  5254 = 'Warnung active'
  160 = 'Waveform'
  980 = 'Waveform File'
  982 = 'Waveform file'
  983 = 'Waveform req.'
  241 = 'Waveform Update'
  12215 = 'WebStrech calculated'
  1096 = 'WebStrech F. Calc'
  1095 = 'WebStrech F. CANopen'
  1094 = 'WebStrech Factor'
  1093 = 'WebStrech Factor CANopen'
  14157 = 'WebStretchFactor'
  13266 = 'WeuReady'
  6459 = 'wI_NominalSpeed'
  6442 = 'wI_PrintMarkDistance'
  317 = 'wI_PurgeTime'
  318 = 'wI_PurgeWaitTime'
  6465 = 'wI_SheetDetectToMark'
  6425 = 'wI_SheetLength'
  6454 = 'wI_SheetThickness'
  6431 = 'wI_SheetWidth'
  321 = 'wI_WaitValveOn'
  677 = 'Work'
  15392 = 'Worker'
  19928 = 'WorkerCamera'
  4305 = 'WorkerDeformation'
  7307 = 'WorkerDelete'
  4323 = 'WorkerPrint 1'
  9993 = 'WorkerPrint 2'
  8780 = 'WorkerPrint enable'
  10042 = 'WorkerPrint PG: %d'
  6644 = 'WorkerPrint selection: %d'
  2559 = 'WorkerPrint1'
  17071 = 'WorkerPrint2'
  5512 = 'WorkerPrint_fPrintStartOffset'
  13893 = 'WorkerVerify'
  12299 = 'WorkerWeu 1'
  17972 = 'WorkerWeu 2'
  1180 = 'WorkerWeu 3'
  1668 = 'WorkerWeu 4'
  1037 = 'Working distance'
  1040 = 'working distance'
  1041 = 'working range'
  1042 = 'working Tempretaure'
  8216 = 'wO_ConveyorSpeed'
  8231 = 'wO_VarnishQuantity'
  454 = 'WrIdx'
  203 = 'Write'
  1160 = 'Write CSV FILE'
  80 = 'Write Settings'
  350 = 'WriteReq'
  346 = 'WrReq'
  1901 = 'X-Offset'
  154 = 'X-Shift'
  187 = 'X-Shift(Offset)'
  174 = 'X-StartPos'
  886 = 'X0'
  15794 = 'X0: %d'
  1638 = 'x: %0.3f'
  2388 = 'x:%0.3f'
  4503 = 'x=%0.4f'
  6585 = 'x=%d'
  18846 = 'x=%f'
  17127 = 'XD: %d'
  887 = 'XS'
  1122 = 'XShift scaled PG1'
  1123 = 'XShift scaled PG2'
  793 = 'Y Shift'
  3801 = 'Y-Offset'
  1 = 'y-shift'
  155 = 'Y-Shift'
  189 = 'Y-Shift(Offset)'
  5249 = 'y: %0.3f'
  18143 = 'y:%0.3f'
  4527 = 'y=%0.4f'
  16177 = 'y=%d'
  8737 = 'y=%f'
  4637 = 'Zero Balance:'
  542 = 'Zero Scale'
  861 = 'Zoom to caller'
  8214 = '[%%] NeutralFibreFactor'
  6372 = '[%%]NeutralFibreFactor'
  6849 = '[+/-]: %f'
  13426 = '[-] WebStrech calculated'
  4770 = '[-]: %f'
  1136 = '[?]: %f'
  864 = '[Base Speed m/s]: %s'
  111 = '[dpi]: %d'
  865 = '[Factor]: %0.6f'
  103 = '[incr./um]: %0.6f'
  1131 = '[Kp]: %f'
  1097 = '[m/min]: %0.3f'
  1098 = '[m/min]: %f'
  17264 = '[m/s] Max. Speed'
  11491 = '[m/s] Speed'
  409 = '[m/s]: %0.3f'
  10053 = '[m/s]: %0.4f'
  404 = '[m/s]: %0.8f'
  109 = '[m/s]: %f'
  105 = '[mm]: %0.3f'
  434 = '[ms]: %d'
  4812 = '[ms]: %f'
  4403 = '[m]'
  801 = '[m] : %f'
  19619 = '[m] LateralRegister'
  8220 = '[m] Module2ToModule3'
  18328 = '[m] SubstrateLength'
  19359 = '[m] SubstrateThickness'
  118 = '[m]: %f'
  104 = '[pulse/px]: %d'
  119 = '[pulse]: %d'
  9440 = '[Px]'
  416 = '[px]: %d'
  410 = '[p]: %d'
  4778 = '[rev/sec]: %f'
  4795 = '[rev]: %f'
  1128 = '[sec]: %f'
  124 = '[Speed m/s]: %s'
  13566 = '[SubPx]'
  106 = '[SubPx]: %d'
  1133 = '[Tn]: %f'
  856 = '[um/inc]: %0.6f'
  10279 = '[um] : %d'
  1121 = '[um] : %f'
  17520 = '[um] SubstrateThickness'
  6048 = '[] SubstrateThickness'
  12440 = '[µm/inc]: %0.6f'
  6503 = '[µm] SubstrateThickness'
  7367 = '[µm]: %0.6f'
  989 = '[µm]: %d'
  67 = '|'
  16114 = '|- verbose'
  11898 = '|- verbose Mode'
  185 = 'µm: %d'
END_TEXTLIST

// ---- POUs/Products/Ink/InkCirculation/_VISU_InkCirculation.TcVIS
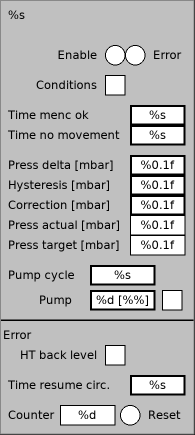
VISUALIZATION _VISU_InkCirculation  // 195x435
VAR_IN_OUT
  m_Inst_Fb : FB_InkCirculation;               (*visu fb instance*) 
END_VAR
    Rectangle (0,0 195x320)
    Rectangle (5,5 180x20), "%s", text variable: m_Inst_Fb._sName
    Ellipse (105,45 20x20), colour toggle: m_Inst_Fb.IbEnable
        toggle m_Inst_Fb.IbEnable
    Rectangle (10,45 90x20), "Enable"
    Ellipse (125,45 20x20), colour toggle: m_Inst_Fb.bLevelError, invisible if: NOT m_Inst_Fb.bLevelError
        toggle m_Inst_Fb.bLevelError
    Rectangle (150,45 40x20), "Error", invisible if: NOT m_Inst_Fb.bLevelError
    Rectangle (5,155 120x20), "Press delta [mbar]"
    Rectangle (130,155 55x20), "%0.1f", text variable: m_Inst_Fb.fRSubMencDeltaP
        OnMouseDown: write the text variable via Edit, min -20, max 0
    Rectangle (5,215 120x20), "Press actual [mbar]"
    Rectangle (130,215 55x20), "%0.1f", text variable: m_Inst_Fb.fSubMencActValue
    Rectangle (5,235 120x20), "Press target [mbar]"
    Rectangle (130,235 55x20), "%0.1f", text variable: m_Inst_Fb.fSubMencTargetValue
    RoundedRectangle (162,290 20x20), colour toggle: m_Inst_Fb.bPumpActivation
    Rectangle (25,290 50x20), "Pump"
    RoundedRectangle (105,75 20x20), colour toggle: m_Inst_Fb.bConditionsMet
    Rectangle (10,75 90x20), "Conditions"
    Rectangle (5,175 120x20), "Hysteresis [mbar]"
    Rectangle (130,175 55x20), "%0.1f", text variable: m_Inst_Fb.fRSubMencHysteresisP
        OnMouseDown: write the text variable via Edit, min 0, max 5
    Rectangle (5,105 120x20), "Time menc ok"
    Rectangle (130,105 55x20), "%s", text variable: m_Inst_Fb.tRSubMencOk
        OnMouseDown: write the text variable via Edit
    Rectangle (5,125 120x20), "Time no movement"
    Rectangle (130,125 55x20), "%s", text variable: m_Inst_Fb.tRNoMovement
        OnMouseDown: write the text variable via Edit
    Rectangle (0,320 195x115)
    Rectangle (0,325 90x20), "Error"
    RoundedRectangle (105,345 20x20), colour toggle: m_Inst_Fb.IbInkLevelReachedBack
    Rectangle (10,345 90x20), "HT back level"
    Rectangle (5,375 120x20), "Time resume circ."
    Rectangle (130,375 55x20), "%s", text variable: m_Inst_Fb.tRResumeCirculation
        OnMouseDown: write the text variable via Edit
    Rectangle (5,405 60x20), "Counter"
    Rectangle (60,405 55x20), "%d", text variable: m_Inst_Fb.nRErrorCounter
    Ellipse (120,405 20x20)
        tap m_Inst_Fb.bResetErrorCounter
    Rectangle (145,405 45x20), "Reset"
    Rectangle (5,195 120x20), "Correction [mbar]"
    Rectangle (130,195 55x20), "%0.1f", text variable: m_Inst_Fb.fRSubMencCorrectionP
        OnMouseDown: write the text variable via Edit, min -1, max 1
    Rectangle (5,265 80x20), "Pump cycle"
    Rectangle (90,265 65x20), "%s", text variable: m_Inst_Fb.tRPumpDutyCycleFrequency
        OnMouseDown: write the text variable via Edit
    Rectangle (90,290 65x20), "%d [%%]", text variable: m_Inst_Fb.nRPumpDutyCycle
        OnMouseDown: write the text variable via Edit
END_VISUALIZATION

// ---- POUs/Products/Machine/_VISU_FUSE_CONTROL.TcVIS
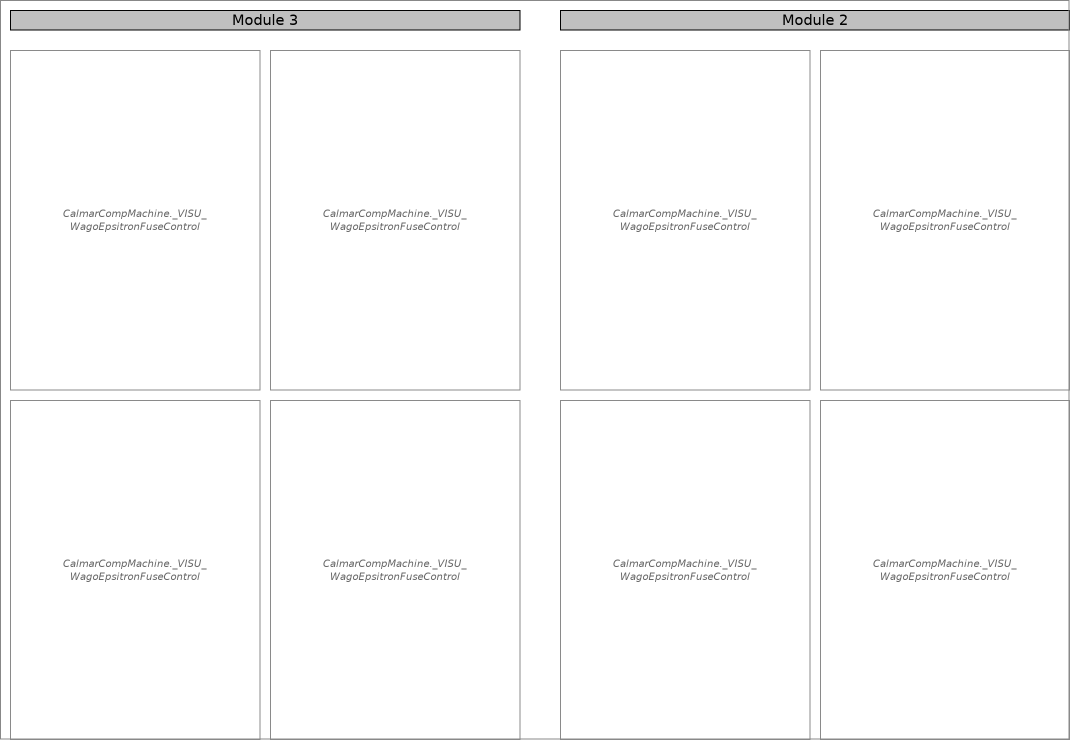
VISUALIZATION _VISU_FUSE_CONTROL  // 1070x740
VAR_IN_OUT
	mInst : FB_WeuPowerControl;
END_VAR
    Frame (820,50 250x340)
        shows CalmarCompMachine._VISU_WagoEpsitronFuseControl(m_Inst_Fb := PRG_MACHINE.fbPowerControl.fb_EpsitronFuseControlF70M1)
    Frame (560,50 250x340)
        shows CalmarCompMachine._VISU_WagoEpsitronFuseControl(m_Inst_Fb := PRG_MACHINE.fbPowerControl.fb_EpsitronFuseControlF90M1)
    Frame (270,50 250x340)
        shows CalmarCompMachine._VISU_WagoEpsitronFuseControl(m_Inst_Fb := PRG_MACHINE.fbPowerControl.fb_EpsitronFuseControlF70M2)
    Frame (10,50 250x340)
        shows CalmarCompMachine._VISU_WagoEpsitronFuseControl(m_Inst_Fb := PRG_MACHINE.fbPowerControl.fb_EpsitronFuseControlF90M2)
    Frame (270,400 250x340), invisible if: TRUE
        shows CalmarCompMachine._VISU_WagoEpsitronFuseControl(m_Inst_Fb := PRG_MACHINE.fbPowerControl.fb_EpsitronFuseControlF122M2)
    Frame (10,400 250x340), invisible if: TRUE
        shows CalmarCompMachine._VISU_WagoEpsitronFuseControl(m_Inst_Fb := PRG_MACHINE.fbPowerControl.fb_EpsitronFuseControlF160M2)
    Frame (820,400 250x340), invisible if: TRUE
        shows CalmarCompMachine._VISU_WagoEpsitronFuseControl(m_Inst_Fb := PRG_MACHINE.fbPowerControl.fb_EpsitronFuseControlF122M1)
    Frame (560,400 250x340), invisible if: TRUE
        shows CalmarCompMachine._VISU_WagoEpsitronFuseControl(m_Inst_Fb := PRG_MACHINE.fbPowerControl.fb_EpsitronFuseControlF160M1)
    Rectangle (10,10 510x20), "Module 3"
    Rectangle (560,10 510x20), "Module 2"
END_VISUALIZATION

// ---- POUs/Products/obsolete/_VISU_DRIFTCONTROL.TcVIS
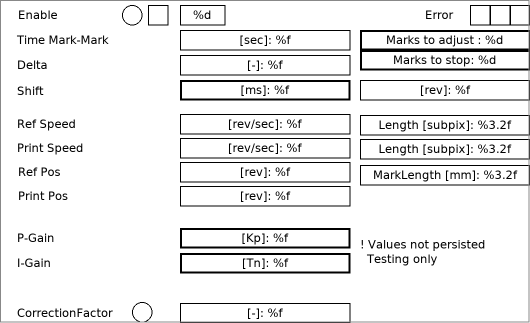
VISUALIZATION _VISU_DRIFTCONTROL  // 530x323
VAR_IN_OUT
  mRef  : FB_DRIFTCONTROL;
END_VAR
    Rectangle (15,5 97x20), "Enable"
    RoundedRectangle (148,5 20x20), colour toggle: mRef.bL_ControlActive
    Ellipse (122,5 20x20), colour toggle: mRef.bI_Enable
        toggle mRef.bI_Enable
    Rectangle (14,30 120x20), "Time Mark-Mark"
    Rectangle (180,30 170x20), "[sec]: %f", text variable: mRef.fL_DeltaTimeStamp
    Rectangle (14,55 120x20), "Delta"
    Rectangle (180,55 170x20), "[-]: %f", text variable: mRef.fL_DeltaCtrl
    Rectangle (14,228 120x20), "P-Gain"
    Rectangle (180,228 170x20), "[Kp]: %f", text variable: mRef.fI_ControllerPGain
        OnMouseDown: write the text variable via Default
    Rectangle (14,253 120x20), "I-Gain"
    Rectangle (180,253 170x20), "[Tn]: %f", text variable: mRef.fI_ControllerIGain
        OnMouseDown: write the text variable via Edit
    Rectangle (14,303 120x20), "CorrectionFactor"
    Rectangle (180,303 170x20), "[-]: %f", text variable: mRef.fO_SpeedCorrectionFactor
    Rectangle (14,114 120x20), "Ref Speed"
    Rectangle (180,114 170x20), "[rev/sec]: %f", text variable: mRef.fL_RefSpeed
    Rectangle (14,138 120x20), "Print Speed"
    Rectangle (180,138 170x20), "[rev/sec]: %f", text variable: mRef.fL_ImgSpeed
    Ellipse (132,302 20x20), colour toggle: mRef.bI_OutputEnable
        toggle mRef.bI_OutputEnable
    Rectangle (360,115 170x20), "Length [subpix]: %3.2f", text variable: mRef.fL_RefLength, colour toggle: mRef.bL_FormatWarning
    Rectangle (360,139 170x20), "Length [subpix]: %3.2f", text variable: mRef.lL_ImgLength, colour toggle: mRef.bL_FormatWarning
    Rectangle (15,162 120x20), "Ref Pos"
    Rectangle (180,162 170x20), "[rev]: %f", text variable: mRef.fL_RefPos
    Rectangle (15,186 120x20), "Print Pos"
    Rectangle (180,186 170x20), "[rev]: %f", text variable: mRef.fL_ImgPos
    RoundedRectangle (470,5 20x20), tooltip "ctrl err", colour toggle: mRef.bO_ContrErr
        tap mRef.bL_ResetInternal
    Rectangle (422,5 42x20), "Error"
    Rectangle (357,233 141x38), "! Values not persisted Testing only"
    Rectangle (180,80 170x20), "[ms]: %f", text variable: mRef.fI_DriftTimeShift
        OnMouseDown: write the text variable via Default
    Rectangle (14,81 120x20), "Shift"
    Rectangle (360,80 170x20), "[rev]: %f", text variable: mRef.fL_ShiftPos
    Rectangle (180,5 45x20), "%d", text variable: mRef.iL_State
    RoundedRectangle (490,5 20x20), tooltip "fb err", colour toggle: mRef.bL_Error
        tap mRef.bL_ResetInternal
    RoundedRectangle (510,5 20x20), tooltip "arw", colour toggle: mRef.fL_CtrlGainFactor <> 1
        tap mRef.bL_ResetInternal
    Rectangle (360,165 170x20), "MarkLength [mm]: %3.2f", text variable: mRef.fL_RefLengthMM, colour toggle: mRef.bL_FormatWarning
    Rectangle (360,30 170x20), "Marks to adjust : %d", text variable: mRef.nI_NbCyclesToAdjust, colour toggle: mRef.bO_ControllerAdjusted
        OnMouseDown: write the text variable via Default
    Rectangle (360,50 170x20), "Marks to stop: %d", text variable: mRef.nI_NbMissMarksToStop, colour toggle: mRef.bO_ControllerAdjusted
        OnMouseDown: write the text variable via Default
END_VISUALIZATION

// ---- POUs/Products/Print_Weu/Mark/_VISU_CameraTrigger.TcVIS
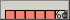
VISUALIZATION _VISU_CameraTrigger  // 70x20
VAR_IN_OUT
	mInst : FB_MarkDetection;
END_VAR
    RoundedRectangle (0,0 70x20), tooltip "Trigger Armed", colour toggle: mInst.bTriggerArmed
    RoundedRectangle (15,10 10x10), tooltip "Speed valid", colour toggle: mInst.bSpeedValid
    RoundedRectangle (25,10 10x10), tooltip "Cam valid", colour toggle: mInst.bCamValid
    RoundedRectangle (35,10 10x10), tooltip "marks valid", colour toggle: mInst.bMarkValid
    RoundedRectangle (5,10 10x10), tooltip "Init ok", colour toggle: mInst.bInitOk
    Rectangle (0,0 70x10), tooltip "Trigger active"
    RoundedRectangle (55,10 10x10), "%d", tooltip "e state", text variable: mInst.nMarkSelection
    RoundedRectangle (45,10 10x10), tooltip "(Hw)Enable", colour toggle: mInst.bEnable
END_VISUALIZATION

// ---- POUs/Products/Print_Weu/Mark/_VISU_MarkCamera_WEU.TcVIS
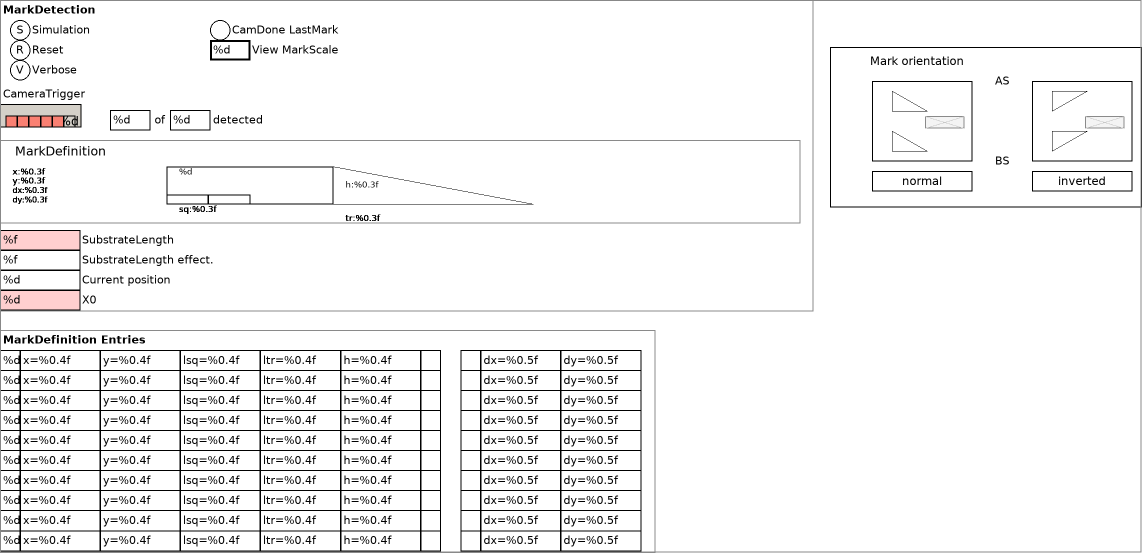
VISUALIZATION _VISU_MarkCamera_WEU  // 1142x553
VAR_IN_OUT
  mCam : FB_MarkCamera_WEU;
  mMarkDetect : FB_MarkDetection;
END_VAR
    Frame (0,330 655x223)
        shows _VISU_MarkDefinition(mInst := mMarkDetect._pFbMarkDefinition^)
    Frame (0,0 813x311)
        shows _VISU_MarkDetection(mInst := mMarkDetect)
    Rectangle (830,47 312x160)
    Rectangle (867,51 124x20), "Mark orientation"
    Rectangle (872,81 100x80)
    Polygon (892,91) (892,111) (927,111)
    Polygon (892,131) (892,151) (927,151)
    Image (925,116 39x12), image: VisuSymbols.Symbols.ArrowBoldLeft
    Rectangle (992,71 25x20), "AS"
    Rectangle (992,151 25x20), "BS"
    Rectangle (1032,81 100x80)
    Polygon (1052,91) (1052,111) (1087,91)
    Polygon (1052,131) (1052,151) (1087,131)
    Image (1085,116 39x12), image: VisuSymbols.Symbols.ArrowBoldLeft
    RoundedRectangle (872,171 100x20), "normal"
    RoundedRectangle (1032,171 100x20), "inverted"
END_VISUALIZATION

// ---- POUs/Products/Print_Weu/Mark/_VISU_MarkDefinition.TcVIS
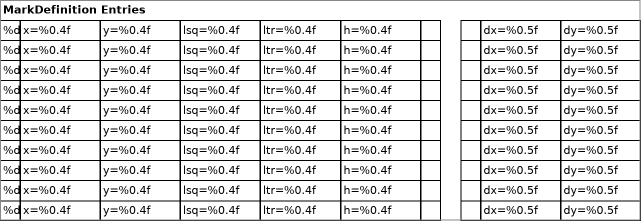
VISUALIZATION _VISU_MarkDefinition  // 641x221
VAR_IN_OUT
	mInst : FB_MarkDefinition;
END_VAR
    Rectangle (0,0 159x20), "MarkDefinition Entries"
    Frame (0,20 641x21)
        shows _VISU_MarkTriangle_Detail(mInst := mInst.sMarkDef[1])
    Frame (0,40 641x21)
        shows _VISU_MarkTriangle_Detail(mInst := mInst.sMarkDef[2])
    Frame (0,60 641x21)
        shows _VISU_MarkTriangle_Detail(mInst := mInst.sMarkDef[3])
    Frame (0,80 641x21)
        shows _VISU_MarkTriangle_Detail(mInst := mInst.sMarkDef[4])
    Frame (0,100 641x21)
        shows _VISU_MarkTriangle_Detail(mInst := mInst.sMarkDef[5])
    Frame (0,200 641x21)
        shows _VISU_MarkTriangle_Detail(mInst := mInst.sMarkDef[10])
    Frame (0,120 641x21)
        shows _VISU_MarkTriangle_Detail(mInst := mInst.sMarkDef[6])
    Frame (0,140 641x21)
        shows _VISU_MarkTriangle_Detail(mInst := mInst.sMarkDef[7])
    Frame (0,160 641x21)
        shows _VISU_MarkTriangle_Detail(mInst := mInst.sMarkDef[8])
    Frame (0,180 641x21)
        shows _VISU_MarkTriangle_Detail(mInst := mInst.sMarkDef[9])
END_VISUALIZATION

// ---- POUs/Products/Print_Weu/Mark/_VISU_MarkDefinition_View.TcVIS
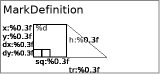
VISUALIZATION _VISU_MarkDefinition_View  // 160x74
VAR_IN_OUT
	mInst : FB_MarkDefinition;
  xScale : UDINT;
END_VAR
    Frame (0,24 160x50), invisible if: NOT mInst.sMarkDef[1].bShow
        shows _VISU_MarkTriangle(mInst := mInst.sMarkDef[1])
        p3560616238: mInst.sMarkDef[1].nMove*xScale
    Frame (0,24 160x50), invisible if: NOT mInst.sMarkDef[2].bShow
        shows _VISU_MarkTriangle(mInst := mInst.sMarkDef[2])
        p3560616238: mInst.sMarkDef[2].nMove*xScale
    Frame (0,24 160x50), invisible if: NOT mInst.sMarkDef[3].bShow
        shows _VISU_MarkTriangle(mInst := mInst.sMarkDef[3])
        p3560616238: mInst.sMarkDef[3].nMove*xScale
    Frame (0,24 160x50), invisible if: NOT mInst.sMarkDef[6].bShow
        shows _VISU_MarkTriangle(mInst := mInst.sMarkDef[6])
        p3560616238: mInst.sMarkDef[6].nMove*xScale
    Frame (0,24 160x50), invisible if: NOT mInst.sMarkDef[4].bShow
        shows _VISU_MarkTriangle(mInst := mInst.sMarkDef[4])
        p3560616238: mInst.sMarkDef[4].nMove*xScale
    Frame (0,24 160x50), invisible if: NOT mInst.sMarkDef[5].bShow
        shows _VISU_MarkTriangle(mInst := mInst.sMarkDef[5])
        p3560616238: mInst.sMarkDef[5].nMove*xScale
    Frame (0,24 160x50), invisible if: NOT mInst.sMarkDef[7].bShow
        shows _VISU_MarkTriangle(mInst := mInst.sMarkDef[7])
        p3560616238: mInst.sMarkDef[7].nMove*xScale
    Frame (0,24 160x50), invisible if: NOT mInst.sMarkDef[10].bShow
        shows _VISU_MarkTriangle(mInst := mInst.sMarkDef[10])
        p3560616238: mInst.sMarkDef[10].nMove*xScale
    Frame (0,24 160x50), invisible if: NOT mInst.sMarkDef[8].bShow
        shows _VISU_MarkTriangle(mInst := mInst.sMarkDef[8])
        p3560616238: mInst.sMarkDef[8].nMove*xScale
    Frame (0,24 160x50), invisible if: NOT mInst.sMarkDef[9].bShow
        shows _VISU_MarkTriangle(mInst := mInst.sMarkDef[9])
        p3560616238: mInst.sMarkDef[9].nMove*xScale
    Rectangle (0,0 120x20), "MarkDefinition"
END_VISUALIZATION

// ---- POUs/Products/Print_Weu/Mark/_VISU_MarkDefinition_View_edit.TcVIS
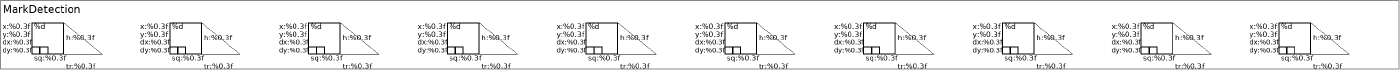
VISUALIZATION _VISU_MarkDefinition_View_edit  // 1463x74
VAR_IN_OUT
	mInst : FB_MarkDefinition;
  xScale : UDINT;
END_VAR
    Frame (0,24 160x50), invisible if: NOT mInst.sMarkDef[1].bShow
        shows _VISU_MarkTriangle(mInst := mInst.sMarkDef[1])
    Frame (144,24 160x50), invisible if: NOT mInst.sMarkDef[2].bShow
        shows _VISU_MarkTriangle(mInst := mInst.sMarkDef[2])
    Frame (289,24 160x50), invisible if: NOT mInst.sMarkDef[3].bShow
        shows _VISU_MarkTriangle(mInst := mInst.sMarkDef[3])
    Frame (724,24 160x50), invisible if: NOT mInst.sMarkDef[6].bShow
        shows _VISU_MarkTriangle(mInst := mInst.sMarkDef[6])
    Frame (434,24 160x50), invisible if: NOT mInst.sMarkDef[4].bShow
        shows _VISU_MarkTriangle(mInst := mInst.sMarkDef[4])
    Frame (579,24 160x50), invisible if: NOT mInst.sMarkDef[5].bShow
        shows _VISU_MarkTriangle(mInst := mInst.sMarkDef[5])
    Frame (869,24 160x50), invisible if: NOT mInst.sMarkDef[7].bShow
        shows _VISU_MarkTriangle(mInst := mInst.sMarkDef[7])
    Frame (1303,24 160x50), invisible if: NOT mInst.sMarkDef[10].bShow
        shows _VISU_MarkTriangle(mInst := mInst.sMarkDef[10])
    Frame (1014,24 160x50), invisible if: NOT mInst.sMarkDef[8].bShow
        shows _VISU_MarkTriangle(mInst := mInst.sMarkDef[8])
    Frame (1159,24 160x50), invisible if: NOT mInst.sMarkDef[9].bShow
        shows _VISU_MarkTriangle(mInst := mInst.sMarkDef[9])
    Rectangle (0,0 120x20), "MarkDetection"
END_VISUALIZATION

// ---- POUs/Products/Print_Weu/Mark/_VISU_MarkDetection.TcVIS
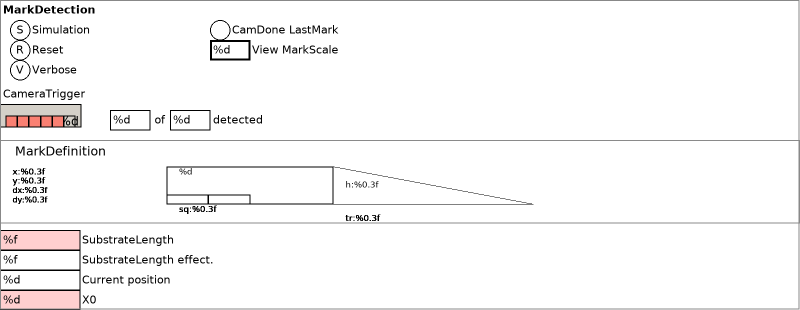
VISUALIZATION _VISU_MarkDetection  // 800x310
VAR_IN_OUT
	mInst: FB_MarkDetection;
END_VAR
    Rectangle (0,0 120x20), "MarkDetection"
    Rectangle (170,110 40x20), "%d", tooltip "teached marks", text variable: mInst._pFbMarkDefinition^._nMarks, colour toggle: mInst._pFbMarkDefinition^._nMarks = 0
    Rectangle (110,110 40x20), "%d", tooltip "detected marks", text variable: mInst._pFbMarkDefinition^._nMarksDetected, colour toggle: mInst._pFbMarkDefinition^._nMarksDetected >= mInst._pFbMarkDefinition^._nMarks AND mInst._pFbMarkDefinition^._nMarks > 0
    Ellipse (10,40 20x20), "R", tooltip "Reset"
        tap mInst.bManualReset
    Frame (0,104 81x26)
        shows _VISU_CameraTrigger(mInst := mInst)
    Rectangle (0,84 120x20), "CameraTrigger"
    Rectangle (210,110 60x20), "detected"
    Rectangle (150,110 20x20), "of"
    Rectangle (0,230 80x20), "%f", text variable: mInst._fSubstrateLength, colour toggle: mInst._fSubstrateLength > 0
    Rectangle (79,230 140x20), "SubstrateLength"
    Rectangle (0,250 80x20), "%f", text variable: mInst._fSubstrateLengthEffective
    Rectangle (79,250 140x20), "SubstrateLength effect."
    Rectangle (0,290 80x20), "%d", text variable: mInst._nX0, colour toggle: mInst._bValid
    Rectangle (79,290 140x20), "X0"
    Rectangle (0,270 80x20), "%d", text variable: mInst.nCurrentPos
    Rectangle (79,270 140x20), "Current position"
    Frame (0,140 800x83)
        shows _VISU_MarkDefinition_View(mInst := mInst._pFbMarkDefinition^, xScale := mInst.nMarkXMoveScale)
    Ellipse (10,20 20x20), "S", tooltip "Simulation"
        toggle mInst._bSimEnable
    Rectangle (29,20 140x20), "Simulation"
    Ellipse (210,20 20x20)
        toggle mInst.bR_TerminateLast
    Rectangle (229,20 140x20), "CamDone LastMark"
    Rectangle (210,40 40x20), "%d", text variable: mInst.nMarkXMoveScale
        OnMouseClick: write the text variable via Default
    Rectangle (249,40 100x20), "View MarkScale"
    Rectangle (29,40 140x20), "Reset"
    Ellipse (10,60 20x20), "V", tooltip "Verbose"
        toggle mInst._bVerbose
    Rectangle (29,60 140x20), "Verbose"
END_VISUALIZATION

// ---- POUs/Products/Print_Weu/Mark/_VISU_MarkTriangle.TcVIS
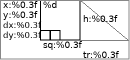
VISUALIZATION _VISU_MarkTriangle  // 130x60
VAR_IN_OUT
	mInst : ST_MarkDefinition;
END_VAR
    Rectangle (40,0 40x40), colour toggle: mInst.sState.bSet
        p874137650: mInst.fSqLength/mInst.fHeight*40-40
    Polygon (80,0) (80,40) (128,40), colour toggle: mInst.sState.bSet
        p3560616238: mInst.fSqLength/mInst.fHeight*40-40
    Rectangle (80,9 40x20), "h:%0.3f", tooltip "[m]", text variable: mInst.fHeight
        p3560616238: mInst.fSqLength/mInst.fHeight*40-40
    Rectangle (80,50 50x10), "tr:%0.3f", tooltip "[m]", text variable: mInst.fTrLength
        p3560616238: mInst.fSqLength/mInst.fHeight*40-40
    Rectangle (40,40 50x10), "sq:%0.3f", tooltip "[m]", text variable: mInst.fSqLength
    Rectangle (40,0 30x10), "%d", tooltip "Id", text variable: mInst.nId
    Rectangle (0,0 40x10), "x:%0.3f", tooltip "[m]", text variable: mInst.fPosX
    Rectangle (0,10 40x10), "y:%0.3f", tooltip "[m]", text variable: mInst.fPosY
    RoundedRectangle (40,30 10x10), tooltip "Missed", colour toggle: mInst.sState.bMissed, invisible if: NOT mInst.sState.bSet
    RoundedRectangle (50,30 10x10), tooltip "InArea", colour toggle: mInst.sState.bInArea, invisible if: NOT mInst.sState.bSet
    Rectangle (0,20 40x10), "dx:%0.3f", tooltip "[m]", text variable: mInst.sState.dx, invisible if: NOT mInst.sState.bSet
    Rectangle (0,30 40x10), "dy:%0.3f", tooltip "[m]", text variable: mInst.sState.dy, invisible if: NOT mInst.sState.bSet
END_VISUALIZATION

// ---- POUs/Products/Print_Weu/Mark/_VISU_MarkTriangle_Detail.TcVIS
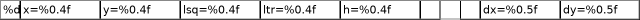
VISUALIZATION _VISU_MarkTriangle_Detail  // 640x20
VAR_IN_OUT
	mInst : ST_MarkDefinition;
END_VAR
    Rectangle (20,0 80x20), "x=%0.4f", text variable: mInst.fPosX
        OnMouseClick: write the text variable via Default
    Rectangle (100,0 80x20), "y=%0.4f", text variable: mInst.fPosY
        OnMouseClick: write the text variable via Default
    RoundedRectangle (460,0 20x20)
        toggle mInst.sState.bSet
    Rectangle (480,0 80x20), "dx=%0.5f", text variable: minst.sState.dx
        OnMouseClick: write the text variable via Default
    Rectangle (560,0 80x20), "dy=%0.5f", text variable: minst.sState.dy
        OnMouseClick: write the text variable via Default
    Rectangle (0,0 20x20), "%d", text variable: mInst.nId, colour toggle: mInst.nId > 0
    RoundedRectangle (420,0 20x20), tooltip "inverted X"
        toggle mInst.bInvertedX
    Rectangle (260,0 80x20), "ltr=%0.4f", text variable: mInst.fTrLength
        OnMouseClick: write the text variable via Default
    Rectangle (340,0 80x20), "h=%0.4f", text variable: mInst.fHeight
        OnMouseClick: write the text variable via Default
    Rectangle (180,0 80x20), "lsq=%0.4f", text variable: mInst.fSqLength
        OnMouseClick: write the text variable via Default
END_VISUALIZATION

// ---- POUs/Products/Print_Weu/UV_LED_Modul/_VISU_UvLedModule.TcVIS
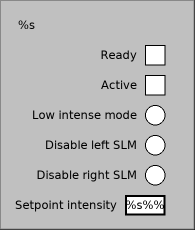
VISUALIZATION _VISU_UvLedModule  // 195x230
VAR_IN_OUT
  m_Inst_Fb   : FB_UvLedModule;
END_VAR
    Rectangle (0,0 195x230), colour variable: m_Inst_Fb._StInkDefinition.lI_ColorRGB
        p2167032090: m_Inst_Fb._StInkDefinition.lI_ColorRGB
        p3092690914: 16#FFFF0000
        p3450524324: 16#FF000000
    Rectangle (15,15 155x20), "%s", text variable: m_Inst_Fb._StInkDefinition.aI_ColorName
    RoundedRectangle (145,45 20x20), colour toggle: m_Inst_Fb.IbReady
    Rectangle (20,45 120x20), "Ready"
    RoundedRectangle (145,75 20x20), colour toggle: m_Inst_Fb._bActivate
    Rectangle (20,75 120x20), "Active"
    Ellipse (145,105 20x20), colour toggle: m_Inst_Fb.RbLowIntenseMode
        toggle m_Inst_Fb.RbLowIntenseMode
    Rectangle (20,105 120x20), "Low intense mode"
    Ellipse (145,135 20x20), colour toggle: m_Inst_Fb.RbDisableLeft
        toggle m_Inst_Fb.RbDisableLeft
    Rectangle (20,135 120x20), "Disable left SLM"
    Ellipse (145,165 20x20), colour toggle: m_Inst_Fb.RbDisableRight
        toggle m_Inst_Fb.RbDisableRight
    Rectangle (20,165 120x20), "Disable right SLM"
    Rectangle (11,195 109x20), "Setpoint intensity"
    Rectangle (125,195 40x20), "%s%%", text variable: m_Inst_Fb.RnIntensitySetpoint
        OnMouseDown: write the text variable via VisuDialogs.Numpad, min m_Inst_Fb.CnMinIntensitySetpoint, max m_Inst_Fb.CnMaxIntensitySetpoint
END_VISUALIZATION

// ---- POUs/Products/Print_Weu/VISU_PAPER_POS_DETECT.TcVIS
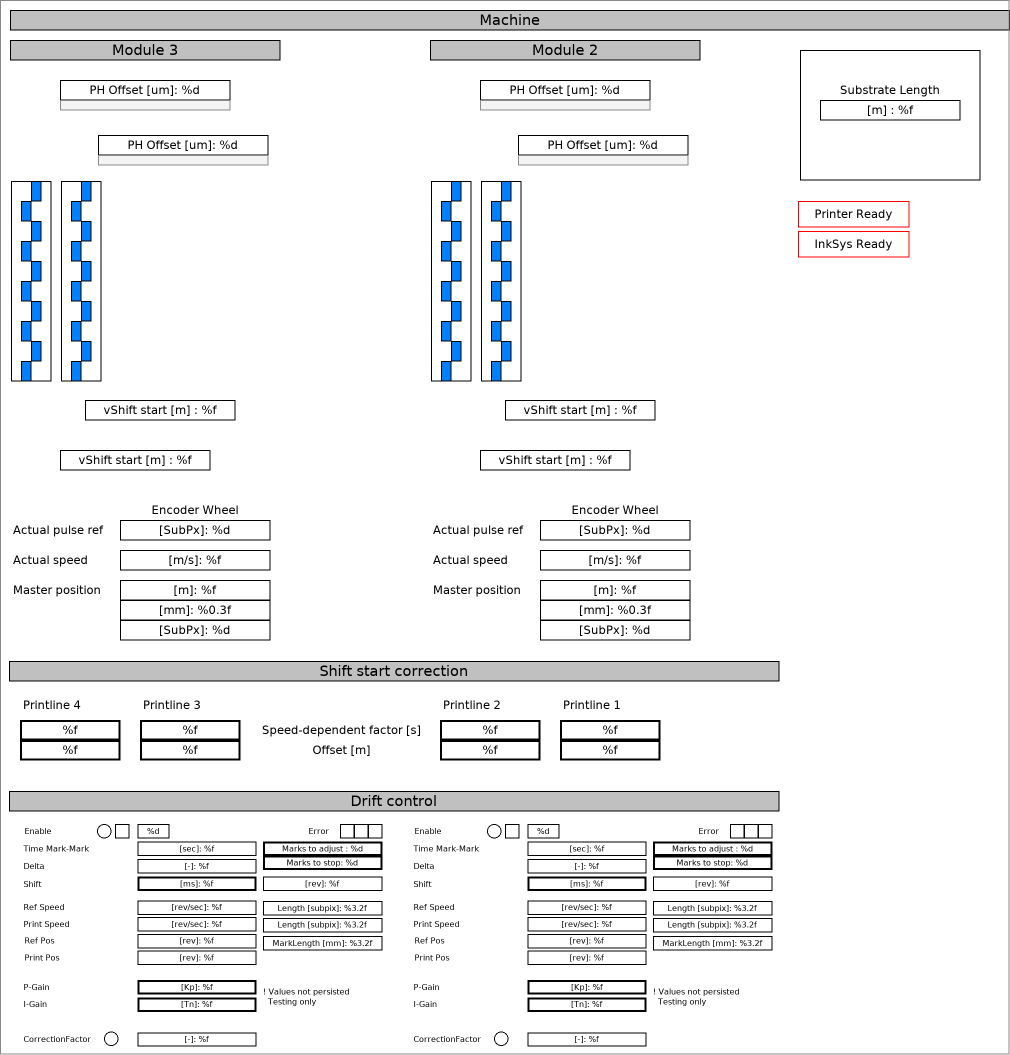
VISUALIZATION VISU_PAPER_POS_DETECT  // 1010x1055
    Polyline (100,340)
    Rectangle (800,50 180x130)
    Rectangle (10,10 1000x20), "Machine"
    Rectangle (820,100 140x20), "[m] : %f", text variable: PRG_PRINT.fL_SubstrateLen[ePr_PG_GROUP_1]
        OnMouseDown: write the text variable via Edit
    Rectangle (820,80 140x20), "Substrate Length"
    Rectangle (798,201 111x26), "Printer Ready", colour toggle: PRG_MACHINE.bO_PrinterReady
    Rectangle (798,231 111x26), "InkSys Ready", colour toggle: PRG_INK.bO_InkSystemOk
    Group (61,181 38x198)
        Rectangle (0,0 40x200)
        Rectangle (20,0 10x20)
        Rectangle (10,20 10x20)
        Rectangle (20,40 10x20)
        Rectangle (10,60 10x20)
        Rectangle (20,80 10x20)
        Rectangle (10,100 10x20)
        Rectangle (20,120 10x20)
        Rectangle (10,140 10x20)
        Rectangle (20,160 10x20)
        Rectangle (10,180 10x20)
    Group (11,181 38x198)
        Rectangle (0,0 40x200)
        Rectangle (20,0 10x20)
        Rectangle (10,20 10x20)
        Rectangle (20,40 10x20)
        Rectangle (10,60 10x20)
        Rectangle (20,80 10x20)
        Rectangle (10,100 10x20)
        Rectangle (20,120 10x20)
        Rectangle (10,140 10x20)
        Rectangle (20,160 10x20)
        Rectangle (10,180 10x20)
    Rectangle (60,80 170x20), "PH Offset [um]: %d", text variable: PRG_PRINT.sAdsPrintGroup[ePr_PG_GROUP_4].sI_ShiftPositionX.lI_Val
        OnMouseDown: write the text variable via Edit
    Scrollbar (60,100 170x10)
        p1057716461: PRG_PRINT.sAdsPrintGroup[ePr_PG_GROUP_2].sI_ShiftPositionX.lI_Val
    Polyline (100,140)
    Polyline (150,360)
    Rectangle (98,135 170x20), "PH Offset [um]: %d", text variable: PRG_PRINT.sAdsPrintGroup[ePr_PG_GROUP_3].sI_ShiftPositionX.lI_Val
        OnMouseDown: write the text variable via Edit
    Scrollbar (98,155 170x10)
        p1057716461: PRG_PRINT.sAdsPrintGroup[ePr_PG_GROUP_1].sI_ShiftPositionX.lI_Val
    Polyline (150,360)
    Polyline (250,350)
    Rectangle (85,400 150x20), "vShift start [m] : %f", text variable: PRG_PRINT.fbWorkerWeu[3].fPosition
    Rectangle (60,450 150x20), "vShift start [m] : %f", text variable: PRG_PRINT.fbWorkerWeu[4].fPosition
    Polyline (100,340)
    Group (481,181 38x198)
        Rectangle (0,0 40x200)
        Rectangle (20,0 10x20)
        Rectangle (10,20 10x20)
        Rectangle (20,40 10x20)
        Rectangle (10,60 10x20)
        Rectangle (20,80 10x20)
        Rectangle (10,100 10x20)
        Rectangle (20,120 10x20)
        Rectangle (10,140 10x20)
        Rectangle (20,160 10x20)
        Rectangle (10,180 10x20)
    Group (431,181 38x198)
        Rectangle (0,0 40x200)
        Rectangle (20,0 10x20)
        Rectangle (10,20 10x20)
        Rectangle (20,40 10x20)
        Rectangle (10,60 10x20)
        Rectangle (20,80 10x20)
        Rectangle (10,100 10x20)
        Rectangle (20,120 10x20)
        Rectangle (10,140 10x20)
        Rectangle (20,160 10x20)
        Rectangle (10,180 10x20)
    Rectangle (480,80 170x20), "PH Offset [um]: %d", text variable: PRG_PRINT.sAdsPrintGroup[ePr_PG_GROUP_2].sI_ShiftPositionX.lI_Val
        OnMouseDown: write the text variable via Edit
    Scrollbar (480,100 170x10)
        p1057716461: PRG_PRINT.sAdsPrintGroup[ePr_PG_GROUP_2].sI_ShiftPositionX.lI_Val
    Polyline (100,140)
    Polyline (150,360)
    Rectangle (518,135 170x20), "PH Offset [um]: %d", text variable: PRG_PRINT.sAdsPrintGroup[ePr_PG_GROUP_1].sI_ShiftPositionX.lI_Val
        OnMouseDown: write the text variable via Edit
    Scrollbar (518,155 170x10)
        p1057716461: PRG_PRINT.sAdsPrintGroup[ePr_PG_GROUP_1].sI_ShiftPositionX.lI_Val
    Polyline (150,360)
    Polyline (250,350)
    Rectangle (505,400 150x20), "vShift start [m] : %f", text variable: PRG_PRINT.fbWorkerWeu[1].fPosition
    Rectangle (480,450 150x20), "vShift start [m] : %f", text variable: PRG_PRINT.fbWorkerWeu[2].fPosition
    Rectangle (10,40 270x20), "Module 3"
    Rectangle (430,40 270x20), "Module 2"
    Rectangle (120,600 150x20), "[mm]: %0.3f", text variable: 0.001*PRG_PRINT.Fb_Ph_Master[ePr_PG_GROUP_2].fO_Master_Position
    Rectangle (120,620 150x20), "[SubPx]: %d", text variable: PRG_PRINT.Fb_Ph_Master[ePr_PG_GROUP_2].lO_Master_Position
    Rectangle (120,550 150x20), "[m/s]: %f", text variable: PRG_PRINT.Fb_Ph_Master[ePr_PG_GROUP_2].fO_Master_Speed
    Rectangle (10,550 100x20), "Actual speed"
    Rectangle (10,580 100x20), "Master position"
    Rectangle (120,520 150x20), "[SubPx]: %d", text variable: PRG_PRINT.Fb_Ph_Master[ePr_PG_GROUP_2].lI_Reference
    Rectangle (10,520 100x20), "Actual pulse ref"
    Rectangle (120,500 150x20), "Encoder Wheel"
    Rectangle (120,580 150x20), "[m]: %f", text variable: 0.000001*PRG_PRINT.Fb_Ph_Master[ePr_PG_GROUP_2].fO_Master_Position
    Rectangle (540,600 150x20), "[mm]: %0.3f", text variable: 0.001*PRG_PRINT.Fb_Ph_Master[ePr_PG_GROUP_1].fO_Master_Position
    Rectangle (540,620 150x20), "[SubPx]: %d", text variable: PRG_PRINT.Fb_Ph_Master[ePr_PG_GROUP_1].lO_Master_Position
    Rectangle (540,550 150x20), "[m/s]: %f", text variable: PRG_PRINT.Fb_Ph_Master[ePr_PG_GROUP_1].fO_Master_Speed
    Rectangle (430,550 100x20), "Actual speed"
    Rectangle (430,580 100x20), "Master position"
    Rectangle (540,520 150x20), "[SubPx]: %d", text variable: PRG_PRINT.Fb_Ph_Master[ePr_PG_GROUP_1].lI_Reference
    Rectangle (430,520 100x20), "Actual pulse ref"
    Rectangle (540,500 150x20), "Encoder Wheel"
    Rectangle (540,580 150x20), "[m]: %f", text variable: 0.000001*PRG_PRINT.Fb_Ph_Master[ePr_PG_GROUP_1].fO_Master_Position
    Frame (12,821 370x234)
        shows _VISU_DRIFTCONTROL(mRef := PRG_PRINT.fB_DriftControl[2])
    Rectangle (9,791 770x20), "Drift control"
    Frame (402,821 370x234)
        shows _VISU_DRIFTCONTROL(mRef := PRG_PRINT.fB_DriftControl[1])
    Rectangle (9,661 770x20), "Shift start correction"
    Rectangle (560,695 100x20), "Printline 1"
    Rectangle (560,720 100x20), "%f", text variable: PRG_PRINT.fbWorkerWeu[1]._fStartShiftFactor
        OnMouseDown: write the text variable via Edit
    Rectangle (560,740 100x20), "%f", text variable: PRG_PRINT.fbWorkerWeu[1]._fStartShiftOffset
        OnMouseDown: write the text variable via Edit
    Rectangle (250,720 180x20), "Speed-dependent factor [s]"
    Rectangle (250,740 180x20), "Offset [m]"
    Rectangle (440,695 100x20), "Printline 2"
    Rectangle (440,720 100x20), "%f", text variable: PRG_PRINT.fbWorkerWeu[2]._fStartShiftFactor
        OnMouseDown: write the text variable via Edit
    Rectangle (440,740 100x20), "%f", text variable: PRG_PRINT.fbWorkerWeu[2]._fStartShiftOffset
        OnMouseDown: write the text variable via Edit
    Rectangle (140,695 100x20), "Printline 3"
    Rectangle (140,720 100x20), "%f", text variable: PRG_PRINT.fbWorkerWeu[3]._fStartShiftFactor
        OnMouseDown: write the text variable via Edit
    Rectangle (140,740 100x20), "%f", text variable: PRG_PRINT.fbWorkerWeu[3]._fStartShiftOffset
        OnMouseDown: write the text variable via Edit
    Rectangle (20,695 100x20), "Printline 4"
    Rectangle (20,720 100x20), "%f", text variable: PRG_PRINT.fbWorkerWeu[4]._fStartShiftFactor
        OnMouseDown: write the text variable via Edit
    Rectangle (20,740 100x20), "%f", text variable: PRG_PRINT.fbWorkerWeu[4]._fStartShiftOffset
        OnMouseDown: write the text variable via Edit
END_VISUALIZATION

// ---- POUs/Products/Print_Weu/_VISU_Templates/_VISU_CT_Details.TcVIS
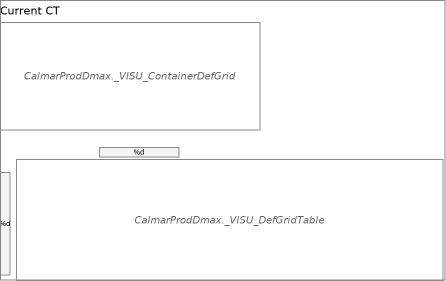
VISUALIZATION _VISU_CT_Details  // 446x281
VAR_IN_OUT
  mInst : FB_WorkerDefGrid_Deformation;
END_VAR
    Frame (0,22 260x108)
        shows CalmarProdDmax._VISU_ContainerDefGrid(m_Inst := mInst._pMultiAttachedCTs[1]^)
    Frame (16,159 427x122)
        shows CalmarProdDmax._VISU_DefGridTable(m_Inst := mInst._pMultiAttachedCTs[1]^.fBImageDeformation, m_row_start := mInst.nGridRowStart, m_col_start := mInst.nGridColStart)
    Scrollbar (99,147 80x10), "%d", text variable: mInst.nGridColStart
        p2245068023: mInst._pMultiAttachedCTs[1]^.fBImageDeformation.nMAX_ROWS_DEFGRID-2
        p1057716461: mInst.nGridColStart
    Scrollbar (0,172 10x103), "%d", text variable: mInst.nGridRowStart
        p2245068023: mInst._pMultiAttachedCTs[1]^.fBImageDeformation.nMAX_ROWS_DEFGRID
        p1057716461: mInst.nGridRowStart
    Label (-3,1 150x20), "Current CT"
END_VISUALIZATION

// ---- POUs/Products/Print_Weu/_VISU_Templates/_VISU_Hardware.TcVIS
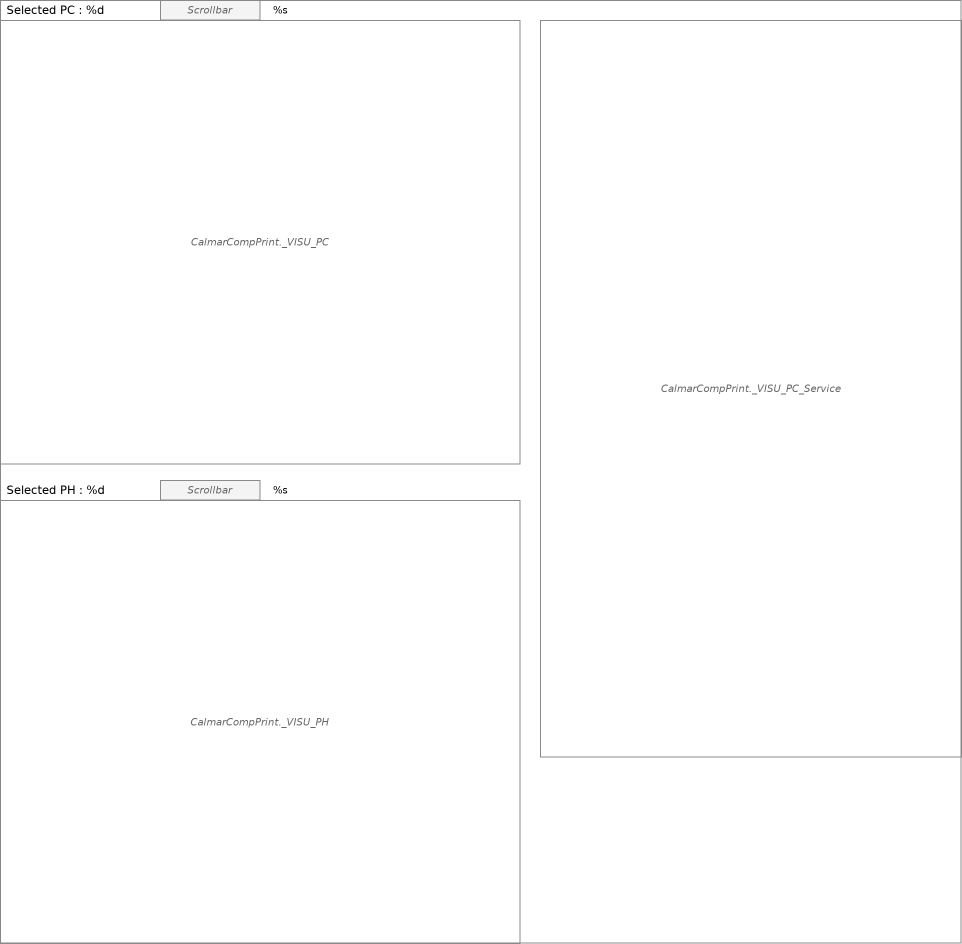
VISUALIZATION _VISU_Hardware  // 962x944
VAR_IN_OUT
	  m_fbHw  : FB_HardwarePool;      (*visu fb instance*)
END_VAR
    Frame (540,20 422x737)
        shows CalmarCompPrint._VISU_PC_Service(m_Inst := m_fbHw._rPcVisuSel^)
    Rectangle (0,0 160x20), "Selected PC : %d", text variable: m_fbHw.fBPcSelector.pSelect^
        OnMouseDown: write the text variable via Edit, min m_fbHw.fBPcSelector.iBoundLower, max m_fbHw.fBPcSelector.iBoundUpper
    Scrollbar (160,0 100x20)
        p3598130195: m_fbHw.fBPcSelector.iBoundLower
        p2245068023: m_fbHw.fBPcSelector.iBoundUpper
        p1057716461: m_fbHw.fBPcSelector.pSelect^
    Rectangle (270,0 250x20), "%s", text variable: m_fbHw._rAdsPcVisuSel^.aO_Name
    Frame (0,20 520x444)
        shows CalmarCompPrint._VISU_PC(m_Inst := m_fbHw._rPcVisuSel^)
    Rectangle (0,480 160x20), "Selected PH : %d", text variable: m_fbHw.fBPhSelector.pSelect^
        OnMouseDown: write the text variable via Edit, min m_fbHw.fBPhSelector.iBoundLower, max m_fbHw.fBPhSelector.iBoundUpper
    Scrollbar (160,480 100x20)
        p3598130195: m_fbHw.fBPhSelector.iBoundLower
        p2245068023: m_fbHw.fBPhSelector.iBoundUpper
        p1057716461: m_fbHw.fBPhSelector.pSelect^
    Rectangle (270,480 250x20), "%s", text variable: m_fbHw._rAdsPhVisuSel^.aO_Name
    Frame (0,500 520x444)
        shows CalmarCompPrint._VISU_PH(m_Inst := m_fbHw._rPhVisuSel^)
END_VISUALIZATION

// ---- POUs/Products/Print_Weu/_VISU_Templates/_VISU_ModuleMaster.TcVIS
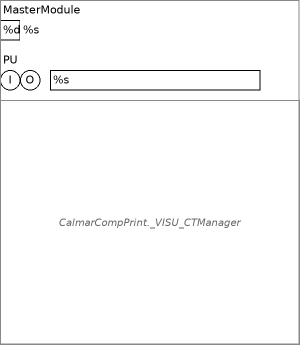
VISUALIZATION _VISU_ModuleMaster  // 300x345
VAR_IN_OUT
	mInst : FB_ModuleMaster;
END_VAR
    Rectangle (50,70 210x20), "%s", tooltip "%s", text variable: mInst._pPU^._activeJob^._sActiveJobDef.sJobSettings.aI_JobName, colour toggle: mInst._pPU^._activeJob <> 0
        p4168582468: mInst._pPU^._activeJob^._sActiveJobDef.sJobSettings.aI_JobName
    Ellipse (0,70 20x20), "I", colour toggle: mInst._pPU^._pAdsPu^.sI_Start.bI_Command OR mInst._pPU^._pAdsPu^.sI_Start.bO_CommandCanEx
        tap mInst._pPU^._pAdsPu^.sI_Start.bI_Command
    Ellipse (20,70 20x20), "O", colour toggle: mInst._pPU^._pAdsPu^.sI_Stop.bI_Command OR mInst._pPU^._pAdsPu^.sI_Stop.bO_CommandCanEx
        tap mInst._pPU^._pAdsPu^.sI_Stop.bI_Command
    Rectangle (0,20 20x20), "%d", tooltip "Master module idx", text variable: mInst._pMasterModule^._nIdx
    Rectangle (0,0 100x20), "MasterModule"
    Rectangle (0,50 100x20), "PU"
    Rectangle (20,20 240x20), "%s", text variable: mInst._pMasterModule^._instanceName
    Frame (0,100 300x245)
        shows CalmarCompPrint._VISU_CTManager(m_Inst := mInst.fBCTManagerMain)
END_VISUALIZATION

// ---- POUs/Products/Print_Weu/_VISU_Templates/_VISU_NeutralFiberDetermine.TcVIS
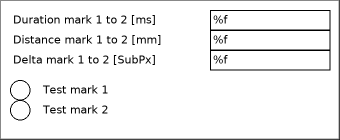
VISUALIZATION _VISU_NeutralFiberDetermine  // 340x140
VAR_IN_OUT
	mInst : FB_NeutralFibreDetermine;
END_VAR
    Rectangle (0,0 340x140)
    Rectangle (10,10 180x20), "Duration mark 1 to 2 [ms]"
    Rectangle (210,10 120x20), "%f", text variable: mInst.fL_DurationMark01to02 / 1000
    Rectangle (10,30 180x20), "Distance mark 1 to 2 [mm]"
    Rectangle (210,30 120x20), "%f", text variable: mInst.fL_LengthMark01to02
        OnMouseClick: write the text variable via Default
    Rectangle (10,50 180x20), "Delta mark 1 to 2 [SubPx]"
    Rectangle (210,50 120x20), "%f", text variable: mInst.nL_DeltaMark01to02
        OnMouseClick: write the text variable via Default
    Ellipse (10,80 20x20), tooltip "Sim VEncoder"
        tap mInst.bIKp_MarkTrigger01
    Rectangle (40,80 100x20), "Test mark 1"
    Ellipse (10,100 20x20), tooltip "Sim VEncoder"
        tap mInst.bIKp_MarkTrigger02
    Rectangle (40,100 100x20), "Test mark 2"
END_VISUALIZATION

// ---- POUs/Products/Print_Weu/_VISU_Templates/_VISU_PmEnable.TcVIS
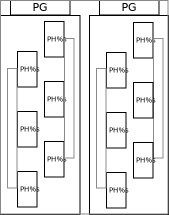
VISUALIZATION _VISU_PmEnable  // 169x215
VAR_IN_OUT
  mInst : FB_PrintModule_Base;
END_VAR
    RoundedRectangle (0,15 80x200), tooltip "WorkerPrint enable"
        toggle mInst.fbWorkerPrint[2]._bEnable
    RoundedRectangle (89,15 80x200), tooltip "WorkerPrint enable"
        toggle mInst.fbWorkerPrint[1]._bEnable
    Rectangle (133,22 20x36)
        toggle mInst._pPh[1]^._pAdsIf^.bI_Enable
    Rectangle (125,30 36x20), angle 270, "PH%s", tooltip "%s", text variable: mInst._pPh[1]^._lIdx
        p4168582468: mInst._pPh[1]^._pAdsIf^.aO_Name
    Frame (153,38 10x120), tooltip "%s"
        shows CalmarCompPrint._VISU_PC_MiniVertical(m_Inst := mInst._pPc[1]^)
        p4168582468: mInst._pPc[1]^._pAds^.aO_Name
    Rectangle (133,82 20x36)
        toggle mInst._pPh[2]^._pAdsIf^.bI_Enable
    Rectangle (133,142 20x36)
        toggle mInst._pPh[3]^._pAdsIf^.bI_Enable
    Rectangle (106,52 20x36)
        toggle mInst._pPh[4]^._pAdsIf^.bI_Enable
    Rectangle (106,112 20x36)
        toggle mInst._pPh[5]^._pAdsIf^.bI_Enable
    Rectangle (106,172 20x36)
        toggle mInst._pPh[6]^._pAdsIf^.bI_Enable
    Rectangle (125,90 36x20), angle 270, "PH%s", tooltip "%s", text variable: mInst._pPh[2]^._lIdx
        p4168582468: mInst._pPh[2]^._pAdsIf^.aO_Name
    Rectangle (125,150 36x20), angle 270, "PH%s", tooltip "%s", text variable: mInst._pPh[3]^._lIdx
        p4168582468: mInst._pPh[3]^._pAdsIf^.aO_Name
    Rectangle (98,60 36x20), angle 270, "PH%s", tooltip "%s", text variable: mInst._pPh[4]^._lIdx
        p4168582468: mInst._pPh[4]^._pAdsIf^.aO_Name
    Rectangle (98,120 36x20), angle 270, "PH%s", tooltip "%s", text variable: mInst._pPh[5]^._lIdx
        p4168582468: mInst._pPh[5]^._pAdsIf^.aO_Name
    Rectangle (98,180 36x20), angle 270, "PH%s", tooltip "%s", text variable: mInst._pPh[6]^._lIdx
        p4168582468: mInst._pPh[6]^._pAdsIf^.aO_Name
    Rectangle (44,21 20x36)
        toggle mInst._pPh[7]^._pAdsIf^.bI_Enable
    Rectangle (36,29 36x20), angle 270, "PH%s", tooltip "%s", text variable: mInst._pPh[7]^._lIdx
        p4168582468: mInst._pPh[7]^._pAdsIf^.aO_Name
    Rectangle (44,81 20x36)
        toggle mInst._pPh[8]^._pAdsIf^.bI_Enable
    Rectangle (44,141 20x36)
        toggle mInst._pPh[9]^._pAdsIf^.bI_Enable
    Rectangle (17,51 20x36)
        toggle mInst._pPh[10]^._pAdsIf^.bI_Enable
    Rectangle (17,111 20x36)
        toggle mInst._pPh[11]^._pAdsIf^.bI_Enable
    Rectangle (17,171 20x36)
        toggle mInst._pPh[12]^._pAdsIf^.bI_Enable
    Rectangle (36,89 36x20), angle 270, "PH%s", tooltip "%s", text variable: mInst._pPh[8]^._lIdx
        p4168582468: mInst._pPh[8]^._pAdsIf^.aO_Name
    Rectangle (36,149 36x20), angle 270, "PH%s", tooltip "%s", text variable: mInst._pPh[9]^._lIdx
        p4168582468: mInst._pPh[9]^._pAdsIf^.aO_Name
    Rectangle (9,59 36x20), angle 270, "PH%s", tooltip "%s", text variable: mInst._pPh[10]^._lIdx
        p4168582468: mInst._pPh[10]^._pAdsIf^.aO_Name
    Rectangle (9,119 36x20), angle 270, "PH%s", tooltip "%s", text variable: mInst._pPh[11]^._lIdx
        p4168582468: mInst._pPh[11]^._pAdsIf^.aO_Name
    Rectangle (9,179 36x20), angle 270, "PH%s", tooltip "%s", text variable: mInst._pPh[12]^._lIdx
        p4168582468: mInst._pPh[12]^._pAdsIf^.aO_Name
    RoundedRectangle (99,0 60x15), "PG", tooltip "PG enable"
        toggle mInst.fbWorkerPrint[1]._pAdsPg^.bI_Enable
    RoundedRectangle (10,0 60x15), "PG", tooltip "PG Enable"
        toggle mInst.fbWorkerPrint[2]._pAdsPg^.bI_Enable
    Frame (96,68 10x120), tooltip "%s"
        shows CalmarCompPrint._VISU_PC_MiniVertical(m_Inst := mInst._pPc[2]^)
        p4168582468: mInst._pPc[1]^._pAds^.aO_Name
    Frame (64,38 10x120), tooltip "%s"
        shows CalmarCompPrint._VISU_PC_MiniVertical(m_Inst := mInst._pPc[3]^)
        p4168582468: mInst._pPc[1]^._pAds^.aO_Name
    Frame (7,68 10x120), tooltip "%s"
        shows CalmarCompPrint._VISU_PC_MiniVertical(m_Inst := mInst._pPc[4]^)
        p4168582468: mInst._pPc[1]^._pAds^.aO_Name
END_VISUALIZATION

// ---- POUs/Products/Print_Weu/_VISU_Templates/_VISU_Pm_Debug.TcVIS
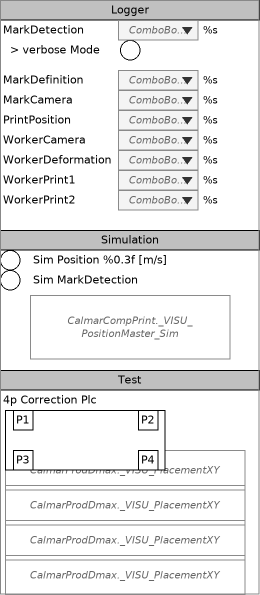
VISUALIZATION _VISU_Pm_Debug  // 260x595
VAR_IN_OUT
	mInst : FB_PrintModule_WEU;
END_VAR
    Rectangle (0,230 260x20), "Simulation"
    Ellipse (0,250 20x20), tooltip "Sim position"
        toggle mInst.fbPrintPosition._bSim
    Rectangle (30,250 200x20), "Sim Position %0.3f [m/s]", text variable: mInst.fbPrintPosition.fbPositionMaster._fSimSpeed
        OnMouseClick: write the text variable via Default
    Ellipse (0,270 20x20), tooltip "Sim position"
        toggle mInst.fbMarkDetection.bSimEnable
    Rectangle (30,270 200x20), "Sim MarkDetection"
    Rectangle (0,0 260x20), "Logger"
    Rectangle (0,20 120x20), "MarkDetection"
    Rectangle (0,70 120x20), "MarkDefinition"
    Rectangle (200,70 60x20), "%s", tooltip "LogLevel", text variable: mInst.fbMarkDefinition._loglevel
        OnMouseClick: write the text variable via Default
    Rectangle (0,90 120x20), "MarkCamera"
    Rectangle (200,90 60x20), "%s", tooltip "LogLevel", text variable: mInst.fbMarkCameraWeu._loglevel
        OnMouseClick: write the text variable via Default
    Rectangle (0,110 120x20), "PrintPosition"
    Rectangle (200,110 60x20), "%s", tooltip "LogLevel", text variable: mInst.fbPrintPosition._loglevel
        OnMouseClick: write the text variable via Default
    Rectangle (0,130 120x20), "WorkerCamera"
    Rectangle (200,130 60x20), "%s", tooltip "LogLevel", text variable: mInst.fbWorkerCamera._loglevel
        OnMouseClick: write the text variable via Default
    Rectangle (0,170 120x20), "WorkerPrint1"
    Rectangle (200,170 60x20), "%s", tooltip "LogLevel", text variable: mInst.fbWorkerPrint[1]._loglevel
        OnMouseClick: write the text variable via Default
    Rectangle (0,190 120x20), "WorkerPrint2"
    Rectangle (200,190 60x20), "%s", tooltip "LogLevel", text variable: mInst.fbWorkerPrint[2]._loglevel
        OnMouseClick: write the text variable via Default
    Rectangle (0,40 120x20), "> verbose Mode"
    Ellipse (120,40 20x20)
        toggle mInst.fbMarkDetection._bVerbose
    Rectangle (0,150 120x20), "WorkerDeformation"
    Rectangle (200,150 60x20), "%s", tooltip "LogLevel", text variable: mInst.fbWorkerDeformation._loglevel
        OnMouseClick: write the text variable via Default
    ComboBoxInteger (118,170 80x20), tooltip "LogLevel", variable: mInst.fbWorkerPrint[1]._loglevel, text list: 'LogSeverity'
    ComboBoxInteger (118,190 80x20), tooltip "LogLevel", variable: mInst.fbWorkerPrint[2]._loglevel, text list: 'LogSeverity'
    ComboBoxInteger (118,150 80x20), tooltip "LogLevel", variable: mInst.fbWorkerDeformation._loglevel, text list: 'LogSeverity'
    ComboBoxInteger (118,130 80x20), tooltip "LogLevel", variable: mInst.fbWorkerCamera._loglevel, text list: 'LogSeverity'
    ComboBoxInteger (118,110 80x20), tooltip "LogLevel", variable: mInst.fbPrintPosition._loglevel, text list: 'LogSeverity'
    ComboBoxInteger (118,90 80x20), tooltip "LogLevel", variable: mInst.fbMarkCameraWeu._loglevel, text list: 'LogSeverity'
    ComboBoxInteger (118,70 80x20), tooltip "LogLevel", variable: mInst.fbMarkDefinition._loglevel, text list: 'LogSeverity'
    Rectangle (200,20 60x20), "%s", tooltip "LogLevel", text variable: mInst.fbMarkDetection._loglevel
        OnMouseClick: write the text variable via Default
    ComboBoxInteger (118,20 80x20), tooltip "LogLevel", variable: mInst.fbMarkDetection._loglevel, text list: 'LogSeverity'
    Frame (30,295 200x64)
        shows CalmarCompPrint._VISU_PositionMaster_Sim(mInst := mInst.fbPrintPosition.fbPositionMaster)
    Frame (5,450 240x40)
        shows CalmarProdDmax._VISU_PlacementXY(m_Inst := mInst.fbFineAlignement._fbPUCorrPoints[1])
    Frame (5,485 240x40)
        shows CalmarProdDmax._VISU_PlacementXY(m_Inst := mInst.fbFineAlignement._fbPUCorrPoints[2])
    Frame (5,520 240x40)
        shows CalmarProdDmax._VISU_PlacementXY(m_Inst := mInst.fbFineAlignement._fbPUCorrPoints[3])
    Frame (5,555 240x40)
        shows CalmarProdDmax._VISU_PlacementXY(m_Inst := mInst.fbFineAlignement._fbPUCorrPoints[4])
    Rectangle (0,390 120x20), "4p Correction Plc"
    Group (5,410 69x30)
        RoundedRectangle (0,0 160x60)
        Rectangle (8,0 20x20), "P1"
        Rectangle (133,0 20x20), "P2"
        Rectangle (133,40 20x20), "P4"
        Rectangle (8,40 20x20), "P3"
    Rectangle (0,370 260x20), "Test"
END_VISUALIZATION

// ---- POUs/Products/Print_Weu/_VISU_Templates/_VISU_Pm_Settings.TcVIS
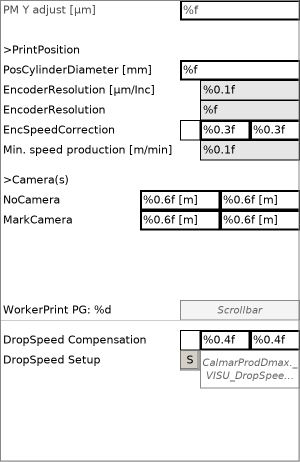
VISUALIZATION _VISU_Pm_Settings  // 300x462
VAR_IN_OUT
	mInst : FB_PrintModule_WEU;
END_VAR
    Rectangle (0,60 180x20), "PosCylinderDiameter [mm]"
    Rectangle (0,80 180x20), "EncoderResolution [µm/Inc]"
    Rectangle (200,80 100x20), "%0.1f", tooltip "constant", text variable: mInst.fC_EncoderImpU
    Rectangle (180,60 120x20), "%f", text variable: mInst._fEncoderCylinderDiameter
        OnMouseClick: write the text variable via Default
    Rectangle (0,0 180x20), "PM Y adjust [µm]"
    Rectangle (180,0 120x20), "%f", text variable: mInst._fPrintModuleAdjustY
        OnMouseClick: write the text variable via VisuDialogs.Numpad, min PRG_PRINT.sC_Config_P.lL_PU_GENERALSHIFT_Y_SET_MIN, max PRG_PRINT.sC_Config_P.lL_PU_GENERALSHIFT_Y_SET_MAX
    Rectangle (250,120 50x20), "%0.3f", tooltip "Encoder speed compensation reference speed", text variable: mInst.fbPrintPosition._fSpeedCompRefSpeed
        OnMouseClick: write the text variable via Default
    Rectangle (200,120 50x20), "%0.3f", tooltip "Encoder speed compensation factor", text variable: mInst.fbPrintPosition._fSpeedCompFactor
        OnMouseClick: write the text variable via Default
    RoundedRectangle (180,120 20x20)
        toggle mInst.fbPrintPosition._bEnSpeedComp
    Rectangle (0,120 180x20), "EncSpeedCorrection"
    Rectangle (0,100 180x20), "EncoderResolution"
    Rectangle (200,100 100x20), "%f", tooltip "by calculation", text variable: mInst.fbPrintPosition._fEncoderResolution
    Scrollbar (180,300 120x20)
        p2245068023: GVL_WEU.nC_WorkerPrintPerPm
        p1057716461: mInst.fbView.nSelWorkerPrint
    Rectangle (0,300 160x20), "WorkerPrint PG: %d", text variable: mInst.fbView.nSelWorkerPrint
    Rectangle (0,320 300x142)
    Rectangle (0,330 180x20), "DropSpeed Compensation"
    Rectangle (200,330 50x20), "%0.4f", tooltip "DropSpeed [m/s]", text variable: mInst.fbWorkerPrint[mInst.fbView.nSelWorkerPrint].fbDropSpeedComp.fDropSpeed
        OnMouseClick: write the text variable via Default
    Rectangle (250,330 50x20), "%0.4f", tooltip "Dead/Add Time [ms]", text variable: mInst.fbWorkerPrint[mInst.fbView.nSelWorkerPrint].fbDropSpeedComp.fDropSpeedDeadTime
        OnMouseClick: write the text variable via Default
    RoundedRectangle (180,330 20x20), tooltip "Enabled compensation", input disabled if: TRUE
        toggle mInst.fbWorkerPrint[mInst.fbView.nSelWorkerPrint].fbDropSpeedComp._bEnable p2164770859=TRUE
    Button (180,350 20x20), "S", tooltip "Setup"
        toggle minst.fbView.bShowDropSpeedSetup
    Rectangle (0,350 180x20), "DropSpeed Setup"
    Frame (200,350 100x38), invisible if: NOT minst.fbView.bShowDropSpeedSetup
        shows CalmarProdDmax._VISU_DropSpeedComp_Setup(mInst := mInst.fbWorkerPrint[mInst.fbView.nSelWorkerPrint].fbDropSpeedComp)
    Rectangle (0,40 180x20), ">PrintPosition"
    Rectangle (0,140 180x20), "Min. speed production [m/min]"
    Rectangle (200,140 100x20), "%0.1f", tooltip "constant", text variable: mInst.fC_ProductionSpeedMpMin_Level
    Rectangle (0,170 180x20), ">Camera(s)"
    Rectangle (220,190 80x20), "%0.6f [m]", tooltip "CameraToPrintUnit", text variable: mInst.fbNoCamera._fCameraToPrintOffset
        OnMouseDown: write the text variable via Default
    Rectangle (140,190 80x20), "%0.6f [m]", tooltip "DetectToCamera", text variable: mInst.fbNoCamera._fDetectToCameraOffset
        OnMouseDown: write the text variable via Default
    Rectangle (0,190 140x20), "NoCamera"
    Rectangle (220,210 80x20), "%0.6f [m]", tooltip "CameraToPrintUnit", text variable: mInst.fbMarkCameraWeu._fCameraToPrintOffset
        OnMouseDown: write the text variable via Default
    Rectangle (140,210 80x20), "%0.6f [m]", tooltip "DetectToCamera", text variable: mInst.fbMarkCameraWeu._fDetectToCameraOffset
        OnMouseDown: write the text variable via Default
    Rectangle (0,210 140x20), "MarkCamera"
END_VISUALIZATION

// ---- POUs/Products/Print_Weu/_VISU_Templates/_VISU_Pm_WEU_bkp.TcVIS
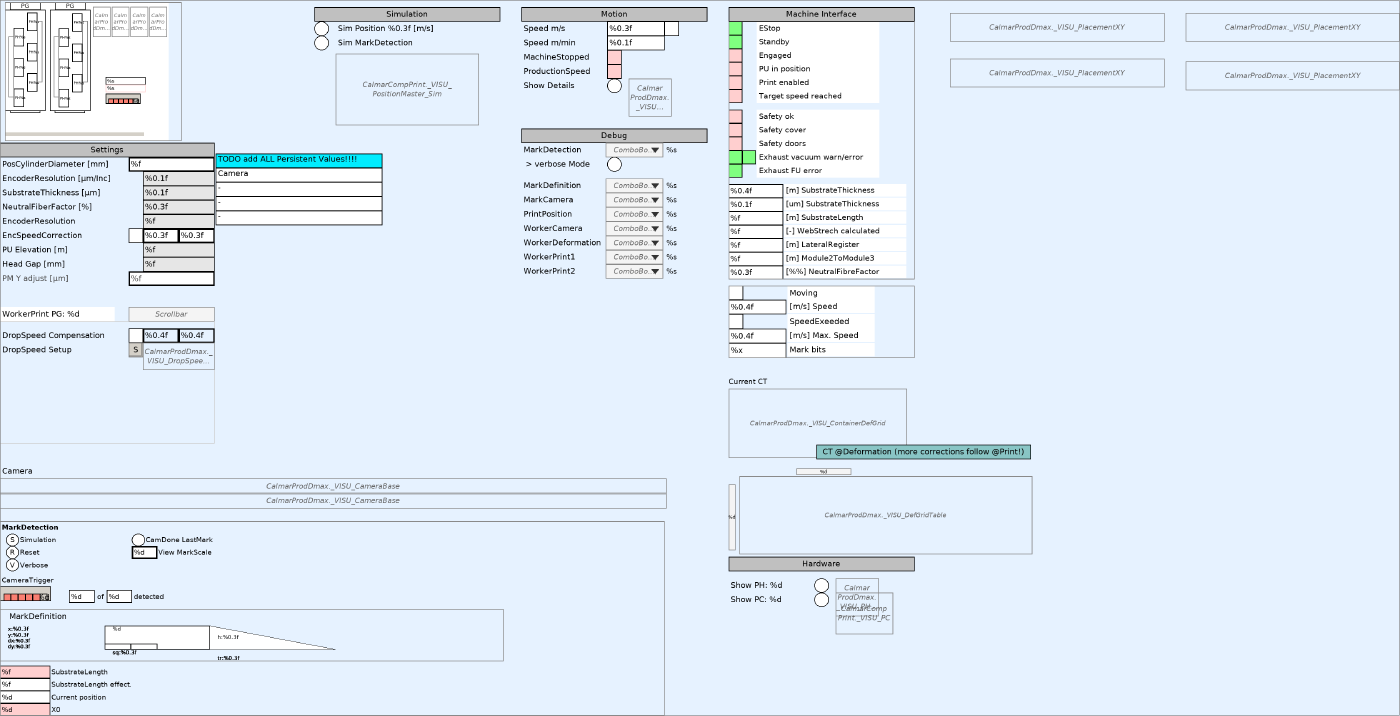
VISUALIZATION _VISU_Pm_WEU_bkp  // 1960x1003
VAR_IN_OUT
  mInst : FB_PrintModule_WEU;
END_VAR
    Rectangle (730,30 120x20), "Speed m/s"
    Rectangle (850,30 80x20), "%0.3f", text variable: mInst.fSpeed
    RoundedRectangle (850,70 20x20), colour toggle: mInst.bMoving
    Rectangle (730,70 110x20), "MachineStopped"
    RoundedRectangle (850,90 20x20), colour toggle: mInst.bProductionSpeedReached
    Rectangle (730,90 110x20), "ProductionSpeed"
    Rectangle (730,50 120x20), "Speed m/min"
    Rectangle (850,50 80x20), "%0.1f", text variable: mInst.fSpeedMpMin
    Rectangle (0,220 180x20), "PosCylinderDiameter [mm]"
    Rectangle (0,240 180x20), "EncoderResolution [µm/Inc]"
    Rectangle (200,240 100x20), "%0.1f", text variable: mInst.fC_EncoderImpU
    Rectangle (180,220 120x20), "%f", text variable: mInst._fEncoderCylinderDiameter
        OnMouseClick: write the text variable via Default
    Rectangle (0,260 180x20), "SubstrateThickness [µm]"
    Rectangle (200,260 100x20), "%0.1f", text variable: mInst._pModuleMachineState^.fSubstrateThickness * 1_000_000
    Rectangle (0,380 180x20), "PM Y adjust [µm]"
    Rectangle (180,380 120x20), "%f", text variable: mInst._fPrintModuleAdjustY
        OnMouseClick: write the text variable via VisuDialogs.Numpad, min PRG_PRINT.sC_Config_P.lL_PU_GENERALSHIFT_Y_SET_MIN, max PRG_PRINT.sC_Config_P.lL_PU_GENERALSHIFT_Y_SET_MAX
    Rectangle (0,360 180x20), "Head Gap [mm]"
    Rectangle (200,360 100x20), "%f", text variable: mInst._pAdsSa^.sI_HeadGap.fI_Val
        OnMouseClick: write the text variable via Default
    RoundedRectangle (930,30 20x20), tooltip "Exeeds max. speed=%f", colour toggle: mInst._pModuleMachineFeedback^.bSpeedExeeded
        p4168582468: mInst._pModuleMachineFeedback^.fMaxSpeed
    Frame (1020,400 260x101)
        shows _VISU_MachineOut(ref := mInst._pModuleMachineFeedback^)
    Frame (1020,30 260x361)
        shows _VISU_MachineIn(ref := mInst._pModuleMachineState^)
    Rectangle (1020,10 260x20), "Machine Interface"
    Rectangle (730,10 260x20), "Motion"
    Frame (0,670 933x22)
        shows CalmarProdDmax._VISU_CameraBase(m_Inst := mInst.fbMarkCameraWeu)
    Frame (0,690 933x22)
        shows CalmarProdDmax._VISU_CameraBase(m_Inst := mInst.fbNoCamera)
    Rectangle (0,650 120x20), "Camera"
    Rectangle (440,10 260x20), "Simulation"
    Ellipse (440,30 20x20), tooltip "Sim position"
        toggle mInst.fbPrintPosition._bSim
    Rectangle (470,30 200x20), "Sim Position %0.3f [m/s]", text variable: mInst.fbPrintPosition.fbPositionMaster._fSimSpeed
        OnMouseClick: write the text variable via Default
    Frame (7,3 247x194)
        shows _VISU_Pm_WEU_mini(mInst := mInst)
    Rectangle (730,110 110x20), "Show Details"
    Ellipse (850,110 20x20)
        toggle mInst.fbView.bShowPositionDetail
    Rectangle (0,200 300x20), "Settings"
    RoundedRectangle (302,235 233x20), "Camera"
    RoundedRectangle (302,255 233x20), "-"
    RoundedRectangle (302,275 233x20), "-"
    RoundedRectangle (302,295 233x20), "-"
    RoundedRectangle (302,215 233x20), "TODO add ALL Persistent Values!!!!"
    Rectangle (250,320 50x20), "%0.3f", tooltip "Encoder speed compensation reference speed", text variable: mInst.fbPrintPosition._fSpeedCompRefSpeed
        OnMouseClick: write the text variable via Default
    Rectangle (200,320 50x20), "%0.3f", tooltip "Encoder speed compensation factor", text variable: mInst.fbPrintPosition._fSpeedCompFactor
        OnMouseClick: write the text variable via Default
    RoundedRectangle (180,320 20x20)
        toggle mInst.fbPrintPosition._bEnSpeedComp
    Rectangle (0,320 180x20), "EncSpeedCorrection"
    Rectangle (0,300 180x20), "EncoderResolution"
    Rectangle (200,300 100x20), "%f", text variable: mInst.fbPrintPosition._fEncoderResolution
    Rectangle (0,280 180x20), "NeutralFiberFactor [%]"
    Rectangle (200,280 100x20), "%0.3f", text variable: mInst._pModuleMachineState^.fNeutralFibreFactor
    Scrollbar (180,430 120x20)
        p2245068023: GVL_WEU.nC_WorkerPrintPerPm
        p1057716461: mInst.fbView.nSelWorkerPrint
    Rectangle (0,430 160x20), "WorkerPrint PG: %d", text variable: mInst.fbView.nSelWorkerPrint
    Rectangle (0,450 300x171)
    Rectangle (0,460 180x20), "DropSpeed Compensation"
    Rectangle (200,460 50x20), "%0.4f", tooltip "DropSpeed [m/s]", text variable: mInst.fbWorkerPrint[mInst.fbView.nSelWorkerPrint].fbDropSpeedComp.fDropSpeed
        OnMouseClick: write the text variable via Default
    Rectangle (250,460 50x20), "%0.4f", tooltip "Dead/Add Time [ms]", text variable: mInst.fbWorkerPrint[mInst.fbView.nSelWorkerPrint].fbDropSpeedComp.fDropSpeedDeadTime
        OnMouseClick: write the text variable via Default
    RoundedRectangle (180,460 20x20), tooltip "Enabled compensation", input disabled if: TRUE
        toggle mInst.fbWorkerPrint[mInst.fbView.nSelWorkerPrint].fbDropSpeedComp._bEnable p2164770859=TRUE
    Button (180,480 20x20), "S", tooltip "Setup"
        toggle minst.fbView.bShowDropSpeedSetup
    Rectangle (0,480 180x20), "DropSpeed Setup"
    Frame (0,730 930x273)
        shows _VISU_MarkDetection(mInst := mInst.fbMarkDetection)
    Ellipse (440,50 20x20), tooltip "Sim position"
        toggle mInst.fbMarkDetection.bSimEnable
    Rectangle (470,50 200x20), "Sim MarkDetection"
    Rectangle (730,180 260x20), "Debug"
    Rectangle (730,200 120x20), "MarkDetection"
    Rectangle (730,250 120x20), "MarkDefinition"
    Rectangle (930,250 60x20), "%s", tooltip "LogLevel", text variable: mInst.fbMarkDefinition._loglevel
        OnMouseClick: write the text variable via Default
    Rectangle (730,270 120x20), "MarkCamera"
    Rectangle (930,270 60x20), "%s", tooltip "LogLevel", text variable: mInst.fbMarkCameraWeu._loglevel
        OnMouseClick: write the text variable via Default
    Rectangle (730,290 120x20), "PrintPosition"
    Rectangle (930,290 60x20), "%s", tooltip "LogLevel", text variable: mInst.fbPrintPosition._loglevel
        OnMouseClick: write the text variable via Default
    Rectangle (730,310 120x20), "WorkerCamera"
    Rectangle (930,310 60x20), "%s", tooltip "LogLevel", text variable: mInst.fbWorkerCamera._loglevel
        OnMouseClick: write the text variable via Default
    Rectangle (730,350 120x20), "WorkerPrint1"
    Rectangle (930,350 60x20), "%s", tooltip "LogLevel", text variable: mInst.fbWorkerPrint[1]._loglevel
        OnMouseClick: write the text variable via Default
    Rectangle (730,370 120x20), "WorkerPrint2"
    Rectangle (930,370 60x20), "%s", tooltip "LogLevel", text variable: mInst.fbWorkerPrint[2]._loglevel
        OnMouseClick: write the text variable via Default
    Frame (200,480 100x38), invisible if: NOT minst.fbView.bShowDropSpeedSetup
        shows CalmarProdDmax._VISU_DropSpeedComp_Setup(mInst := mInst.fbWorkerPrint[mInst.fbView.nSelWorkerPrint].fbDropSpeedComp)
    Frame (880,110 60x53), invisible if: NOT mInst.fbView.bShowPositionDetail
        shows CalmarProdDmax._VISU_PrintPositionDmax(m_Inst := mInst.fbPrintPosition)
    Rectangle (726,220 124x20), "> verbose Mode"
    Ellipse (850,220 20x20)
        toggle mInst.fbMarkDetection._bVerbose
    Frame (1020,525 428x251)
        shows _VISU_CT_Details(mInst := mInst.fbWorkerDeformation)
    Rectangle (730,330 120x20), "WorkerDeformation"
    Rectangle (930,330 60x20), "%s", tooltip "LogLevel", text variable: mInst.fbWorkerDeformation._loglevel
        OnMouseClick: write the text variable via Default
    ComboBoxInteger (848,350 80x20), tooltip "LogLevel", variable: mInst.fbWorkerPrint[1]._loglevel, text list: 'LogSeverity'
    ComboBoxInteger (848,370 80x20), tooltip "LogLevel", variable: mInst.fbWorkerPrint[2]._loglevel, text list: 'LogSeverity'
    ComboBoxInteger (848,330 80x20), tooltip "LogLevel", variable: mInst.fbWorkerDeformation._loglevel, text list: 'LogSeverity'
    ComboBoxInteger (848,310 80x20), tooltip "LogLevel", variable: mInst.fbWorkerCamera._loglevel, text list: 'LogSeverity'
    ComboBoxInteger (848,290 80x20), tooltip "LogLevel", variable: mInst.fbPrintPosition._loglevel, text list: 'LogSeverity'
    ComboBoxInteger (848,270 80x20), tooltip "LogLevel", variable: mInst.fbMarkCameraWeu._loglevel, text list: 'LogSeverity'
    ComboBoxInteger (848,250 80x20), tooltip "LogLevel", variable: mInst.fbMarkDefinition._loglevel, text list: 'LogSeverity'
    Rectangle (930,200 60x20), "%s", tooltip "LogLevel", text variable: mInst.fbMarkDetection._loglevel
        OnMouseClick: write the text variable via Default
    ComboBoxInteger (848,200 80x20), tooltip "LogLevel", variable: mInst.fbMarkDetection._loglevel, text list: 'LogSeverity'
    Ellipse (1140,810 20x20)
        toggle mInst.fbView.bShowPhDetail
    Frame (1170,810 60x53), invisible if: NOT mInst.fbView.bShowPhDetail
        shows CalmarProdDmax._VISU_PH_Grid(m_Inst := mInst._pPh[mInst.fbView.nSelPhDetail]^)
    Rectangle (1020,810 110x20), "Show PH: %d", text variable: mInst.fbView.nSelPhDetail
        OnMouseClick: write the text variable via Default
    Rectangle (1020,780 260x20), "Hardware"
    Ellipse (1140,830 20x20)
        toggle mInst.fbView.bShowPcDetail
    Frame (1170,830 80x58), invisible if: NOT mInst.fbView.bShowPcDetail
        shows CalmarCompPrint._VISU_PC(m_Inst := mInst._pPc[mInst.fbView.nSelPcDetail]^)
    Rectangle (1020,830 110x20), "Show PC: %d", text variable: mInst.fbView.nSelPcDetail
        OnMouseClick: write the text variable via Default
    Rectangle (200,340 100x20), "%f", text variable: mInst.fPuElevation
        OnMouseClick: write the text variable via Default
    Rectangle (0,340 180x20), "PU Elevation [m]"
    Frame (470,75 200x100)
        shows CalmarCompPrint._VISU_PositionMaster_Sim(mInst := mInst.fbPrintPosition.fbPositionMaster)
    Frame (1330,18 300x40)
        shows CalmarProdDmax._VISU_PlacementXY(m_Inst := mInst.fbFineAlignement._fbPUCorrPoints[1])
    Frame (1660,18 300x40)
        shows CalmarProdDmax._VISU_PlacementXY(m_Inst := mInst.fbFineAlignement._fbPUCorrPoints[2])
    Frame (1330,82 300x40)
        shows CalmarProdDmax._VISU_PlacementXY(m_Inst := mInst.fbFineAlignement._fbPUCorrPoints[3])
    Frame (1660,86 300x40)
        shows CalmarProdDmax._VISU_PlacementXY(m_Inst := mInst.fbFineAlignement._fbPUCorrPoints[4])
    Rectangle (1143,623 300x20), "CT @Deformation (more corrections follow @Print!)"
END_VISUALIZATION

// ---- POUs/Products/Print_Weu/_VISU_Templates/_VISU_Pm_WEU_mini.TcVIS
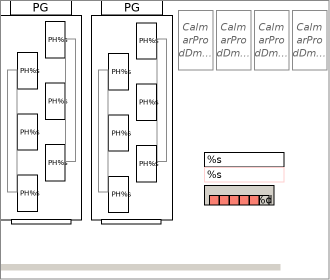
VISUALIZATION _VISU_Pm_WEU_mini  // 330x280
VAR_IN_OUT
  mInst : FB_PrintModule_WEU;
END_VAR
    Rectangle (0,0 330x280)
    Frame (204,185 61x21)
        shows _VISU_CameraTrigger(mInst := mInst.fbMarkDetection)
    Rectangle (204,152 80x15), "%s", tooltip "active camera device", text variable: mInst.fbWorkerCamera._iActiveCam.sName
    Rectangle (204,167 80x15), "%s", tooltip "active camera mode", text variable: mInst.fbWorkerCamera._iActiveCam.eCameraMode, colour toggle: mInst.fbWorkerCamera._bCamValid
    RoundedRectangle (0,264 280x6), colour toggle: mInst.fbView.bMovingInd
    Frame (0,0 177x220)
        shows _VISU_PmEnable(mInst := mInst)
        p2738717112: mInst.fbView.zPos_PM
    RoundedRectangle (11,219 60x5), colour toggle: mInst.fbView.bPrintInd[2]
        p2738717112: mInst.fbView.zPos_PM
    RoundedRectangle (101,219 60x5), colour toggle: mInst.fbView.bPrintInd[1]
        p2738717112: mInst.fbView.zPos_PM
    Line (0,0) (280,0)
    Frame (254,10 35x60)
        shows CalmarProdDmax._VISU_WorkerDefGrid_small(m_Inst := mInst.fbWorkerDeformation)
    Frame (292,10 35x60)
        shows CalmarProdDmax._VISU_WorkerDefGrid_small(m_Inst := mInst.fbWorkerCamera)
    Frame (178,10 35x60)
        shows CalmarProdDmax._VISU_WorkerDefGrid_small(m_Inst := mInst.fbWorkerPrint[2])
    Frame (216,10 35x60)
        shows CalmarProdDmax._VISU_WorkerDefGrid_small(m_Inst := mInst.fbWorkerPrint[1])
END_VISUALIZATION

// ---- POUs/Products/Print_Weu/_VISU_Templates/_VISU_Pm_WEU.TcVIS
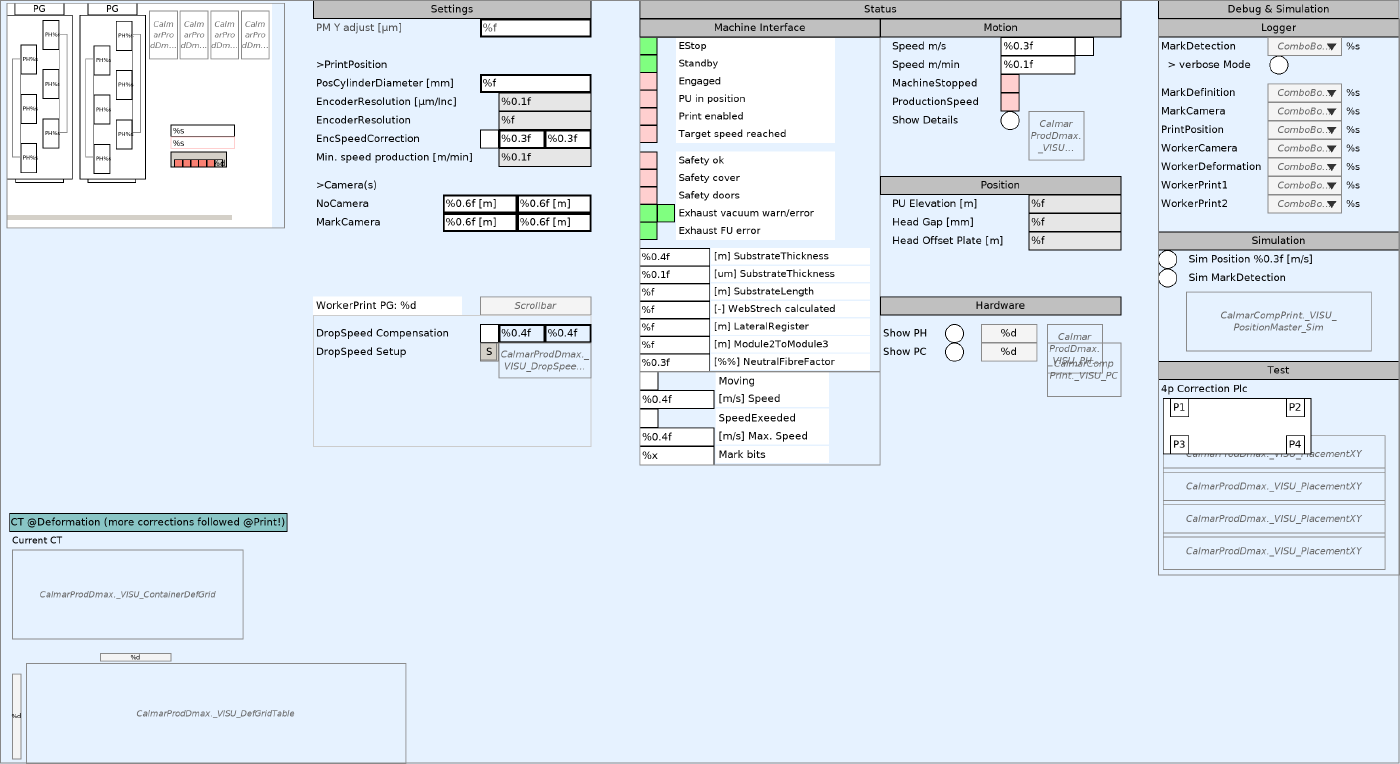
VISUALIZATION _VISU_Pm_WEU  // 1511x825
VAR_IN_OUT
  mInst : FB_PrintModule_WEU;
END_VAR
    Rectangle (960,40 120x20), "Speed m/s"
    Rectangle (1080,40 80x20), "%0.3f", text variable: mInst.fSpeed
    RoundedRectangle (1080,80 20x20), colour toggle: mInst.bMoving
    Rectangle (960,80 110x20), "MachineStopped"
    RoundedRectangle (1080,100 20x20), colour toggle: mInst.bProductionSpeedReached
    Rectangle (960,100 110x20), "ProductionSpeed"
    Rectangle (960,60 120x20), "Speed m/min"
    Rectangle (1080,60 80x20), "%0.1f", text variable: mInst.fSpeedMpMin
    RoundedRectangle (1160,40 20x20), tooltip "Exeeds max. speed=%f", colour toggle: mInst._pModuleMachineFeedback^.bSpeedExeeded
        p4168582468: mInst._pModuleMachineFeedback^.fMaxSpeed
    Frame (690,401 260x101)
        shows _VISU_MachineOut(ref := mInst._pModuleMachineFeedback^)
    Frame (690,40 260x361)
        shows _VISU_MachineIn(ref := mInst._pModuleMachineState^)
    Rectangle (690,20 260x20), "Machine Interface"
    Rectangle (950,20 260x20), "Motion"
    Frame (7,3 300x243)
        shows _VISU_Pm_WEU_mini(mInst := mInst)
    Rectangle (960,120 110x20), "Show Details"
    Ellipse (1080,120 20x20)
        toggle mInst.fbView.bShowPositionDetail
    Frame (13,574 428x251)
        shows _VISU_CT_Details(mInst := mInst.fbWorkerDeformation)
    Ellipse (1020,350 20x20)
        toggle mInst.fbView.bShowPhDetail
    Rectangle (950,350 110x20), "Show PH"
    Rectangle (950,320 260x20), "Hardware"
    Ellipse (1020,370 20x20)
        toggle mInst.fbView.bShowPcDetail
    Rectangle (950,370 110x20), "Show PC"
    Rectangle (10,554 300x20), "CT @Deformation (more corrections followed @Print!)"
    Scrollbar (1059,350 60x20), "%d", text variable: mInst.fbView.nSelPhDetail
        p2245068023: mInst._nPh
        p1057716461: mInst.fbView.nSelPhDetail
    Scrollbar (1059,370 60x20), "%d", text variable: mInst.fbView.nSelPcDetail
        p2245068023: mInst._nPc
        p1057716461: mInst.fbView.nSelPcDetail
    Frame (1250,20 261x601), invisible if: NOT mInst.fbView.bShowDebugAndSim
        shows _VISU_Pm_Debug(mInst := mInst)
    Frame (338,20 299x522)
        shows _VISU_Pm_Settings(mInst := mInst)
    Rectangle (338,0 300x20), "Settings"
    Rectangle (690,0 520x20), "Status"
    Rectangle (1250,0 260x20), "Debug & Simulation"
        toggle mInst.fbView.bShowDebugAndSim
    Rectangle (950,190 260x20), "Position"
    Rectangle (960,230 140x20), "Head Gap [mm]"
    Rectangle (1110,230 100x20), "%f", text variable: mInst._pAdsSa^.sI_HeadGap.fI_Val
    Rectangle (1110,210 100x20), "%f", text variable: mInst.fPuElevation
    Rectangle (960,210 140x20), "PU Elevation [m]"
    Rectangle (960,250 140x20), "Head Offset Plate [m]"
    Rectangle (1110,250 100x20), "%f", text variable: mInst.fC_HeadOffsetPlate
    Frame (1110,120 60x53), invisible if: NOT mInst.fbView.bShowPositionDetail
        shows CalmarProdDmax._VISU_PrintPositionDmax(m_Inst := mInst.fbPrintPosition)
    Frame (1130,350 60x53), invisible if: NOT mInst.fbView.bShowPhDetail
        shows CalmarProdDmax._VISU_PH_Grid(m_Inst := mInst._pPh[mInst.fbView.nSelPhDetail]^)
    Frame (1130,370 80x58), invisible if: NOT mInst.fbView.bShowPcDetail
        shows CalmarCompPrint._VISU_PC(m_Inst := mInst._pPc[mInst.fbView.nSelPcDetail]^)
END_VISUALIZATION

// ---- POUs/Products/Print_Weu/_VISU_Templates/_VISU_WorkerPrint_WEU.TcVIS
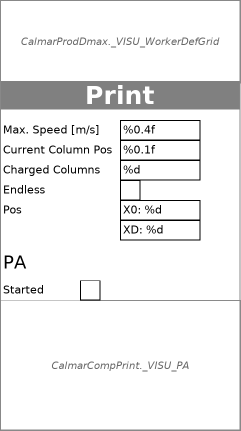
VISUALIZATION _VISU_WorkerPrint_WEU  // 241x431
VAR_IN_OUT
  m_Inst : FB_WorkerDefGrid_Print_WEU;
END_VAR
    Frame (0,0 241x83)
        shows CalmarProdDmax._VISU_WorkerDefGrid(m_Inst := m_Inst)
    Rectangle (0,80 240x30), "Print", colour toggle: m_Inst._pAttachedCt <> 0
    Frame (0,300 241x131)
        shows CalmarCompPrint._VISU_PA(m_Inst := m_Inst.fbPa)
    Rectangle (0,120 120x20), "Max. Speed [m/s]"
    Rectangle (120,120 80x20), "%0.4f", text variable: m_Inst.fMaxSpeed
    Rectangle (0,140 120x20), "Current Column Pos"
    Rectangle (120,140 80x20), "%0.1f", text variable: m_Inst.fCurrentColumnPos
    Rectangle (0,160 120x20), "Charged Columns"
    Rectangle (120,160 80x20), "%d", text variable: m_Inst.nChargedColumns
    Rectangle (0,180 120x20), "Endless"
    RoundedRectangle (120,180 20x20), colour toggle: m_Inst._bEndless
    Rectangle (0,280 80x20), "Started"
    RoundedRectangle (80,280 20x20), colour toggle: m_Inst._bPaStarted
    Rectangle (0,200 120x20), "Pos"
    Rectangle (120,200 80x20), "X0: %d", text variable: m_Inst._nPosX0
    Rectangle (120,220 80x20), "XD: %d", text variable: m_Inst._nPosXDelta
    Rectangle (0,250 240x30), "PA"
END_VISUALIZATION

// ---- POUs/Products/Print_Weu/_VISU_Templates/_VISU_Pm_Worker.TcVIS
